(* PLC project Система умного дома.project, CODESYS CODESYS V3.5 SP17 Patch 3 *)
(* stored: creationDateTime 2026-04-06T20:38:17.5908527, modificationDateTime 2026-03-25T09:46:39.3897592 *)

TYPE E_ALERT_PRIORITY : (ALERT_PRIORITY_NONE := 0, ALERT_PRIORITY_LOW := 1, ALERT_PRIORITY_MEDIUM := 2, ALERT_PRIORITY_HIGH := 3, ALERT_PRIORITY_CRITICAL := 4) USINT;
END_TYPE

TYPE E_Debug_Log_Level : (LOG_LEVEL_MINIMAL := 0, LOG_LEVEL_NORMAL := 1, LOG_LEVEL_VERBOSE := 2, LOG_LEVEL_DEBUG := 3) USINT;
END_TYPE

TYPE E_Gateway_Command_Type : (CMD_NONE := 0, CMD_SET_SCENARIO := 1, CMD_SET_LIGHT := 2, CMD_SET_SOCKET := 3, CMD_SET_SECURITY := 4, CMD_SET_TEMP := 5, CMD_SET_VENT := 6, CMD_SET_BLINDS := 7, CMD_TELEGRAM_MSG := 8) USINT;
END_TYPE

TYPE E_Lifetime_Device_Type : (LIFETIME_DEVICE_PUMP := 1, LIFETIME_DEVICE_FAN := 2) USINT;
END_TYPE

TYPE E_Outdoor_Mode : (OUTDOOR_MODE_AUTO := 0, OUTDOOR_MODE_PARTY := 1, OUTDOOR_MODE_SECURITY := 2, OUTDOOR_MODE_ECONOMY := 3, OUTDOOR_MODE_MANUAL := 4) USINT;
END_TYPE

TYPE E_PLC_ROLE : (ROLE_UNDEFINED := 0, ROLE_ACTIVE := 1, ROLE_STANDBY := 2, ROLE_OFFLINE := 3) USINT;
END_TYPE

TYPE E_Rule_Action_Type : (ACTION_NONE := 0, ACTION_SET_FLOOR_HEATING := 1, ACTION_SET_LIGHTING_BASE := 2, ACTION_SET_LIGHTING_ACCENT := 3, ACTION_SET_SOCKET := 4, ACTION_SET_VENTILATION := 5, ACTION_SET_BLINDS := 6, ACTION_ACTIVATE_SCENARIO := 7, ACTION_TOGGLE_LIGHTING := 8, ACTION_TOGGLE_SOCKET := 9) USINT;
END_TYPE

TYPE E_Rule_Comparison : (COMP_NONE := 0, COMP_EQ := 1, COMP_GT := 2, COMP_LT := 3, COMP_GE := 4, COMP_LE := 5, COMP_IN_RANGE := 6, COMP_TRUE := 7, COMP_FALSE := 8) USINT;
END_TYPE

TYPE E_Rule_Condition_Type : (COND_NONE := 0, COND_AIR_TEMP := 1, COND_FLOOR_TEMP := 2, COND_HUMIDITY := 3, COND_CO2 := 4, COND_METHANE := 5, COND_CO := 6, COND_DOOR_WINDOW := 7, COND_FLOOD := 8, COND_SMOKE := 9, COND_MOTION := 10, COND_TIME_OF_DAY := 11, COND_DAY_OF_WEEK := 12) USINT;
END_TYPE

TYPE E_SCENARIO_TYPE : (SCENARIO_NONE := 0, SCENARIO_MORNING := 1, SCENARIO_EVENING := 2, SCENARIO_AWAY := 3, SCENARIO_PARTY := 4, SCENARIO_SLEEP := 5, SCENARIO_EMERGENCY := 6, SCENARIO_PRESENCE := 7) USINT;
END_TYPE

TYPE E_SENSOR_TYPE : (SENSOR_TYPE_NONE := 0, SENSOR_TYPE_DOOR_WINDOW := 5, SENSOR_TYPE_GLASS_BREAK := 6, SENSOR_TYPE_FLOOD := 7, SENSOR_TYPE_SMOKE := 8, SENSOR_TYPE_GAS_METHANE := 1, SENSOR_TYPE_GAS_CO := 2, SENSOR_TYPE_TEMP_FLOOR := 3, SENSOR_TYPE_TEMP_AIR := 4, SENSOR_TYPE_CO2 := 9) USINT;
END_TYPE

TYPE E_System_Operating_Mode : (MODE_NORMAL := 0, MODE_DEGRADED := 1, MODE_SAFE_STOP := 2, MODE_FREEZE_PROTECTION := 3) INT;
END_TYPE

TYPE E_System_Root_Cause : (ROOT_NONE := 0, ROOT_FIRE := 1, ROOT_GAS_LEAK := 2, ROOT_CO_WARNING := 3, ROOT_CO_CRITICAL := 4, ROOT_WATER_LEAK := 5, ROOT_IO_OFFLINE := 6, ROOT_COMM_FAULT := 7, ROOT_SENSOR_FAULT := 8, ROOT_SUBSYSTEM_FAULT := 9, ROOT_WATCHDOG_FAULT := 10) INT;
END_TYPE

TYPE E_System_Severity : (SEV_NORMAL := 0, SEV_WARNING := 1, SEV_DEGRADED := 2, SEV_CRITICAL := 3) INT;
END_TYPE

TYPE E_Trend_Parameter_Type : (TREND_PARAM_NONE := 0, TREND_PARAM_TEMP_AIR := 1, TREND_PARAM_TEMP_FLOOR := 2, TREND_PARAM_PRESSURE := 3, TREND_PARAM_PUMP_CURRENT := 4, TREND_PARAM_GAS_METHANE := 5, TREND_PARAM_GAS_CO := 6) USINT;
END_TYPE

TYPE E_TwoFactor_Method : (TF_METHOD_NONE := 0, TF_METHOD_RFID := 1, TF_METHOD_TOTP := 2, TF_METHOD_BOTH := 3) USINT;
END_TYPE

TYPE E_VALVE_TYPE : (VALVE_NC := 1, VALVE_NO := 2) USINT;
END_TYPE

TYPE E_VENTILATION_LOCATION : (VENT_LOCATION_NONE := 0, VENT_LOCATION_BASEMENT_GAME_ROOM := 1, VENT_LOCATION_BASEMENT_GYM := 2, VENT_LOCATION_BASEMENT_BOILER_ROOM := 3, VENT_LOCATION_BATHROOM_1F := 4, VENT_LOCATION_BATHROOM_2F := 5, VENT_LOCATION_MASTER_BATHROOM := 6, VENT_LOCATION_LAUNDRY := 7, VENT_LOCATION_KITCHEN := 8) USINT;
END_TYPE

TYPE E_VENTILATION_UNIT_TYPE : (VENTILATION_TYPE_NONE := 0, VENTILATION_TYPE_SUPPLY := 1, VENTILATION_TYPE_EXHAUST := 2) USINT;
END_TYPE

TYPE E_Valve_Test_Result : (TEST_RESULT_NONE := 0, TEST_RESULT_PASSED := 1, TEST_RESULT_CURRENT_DEVIATION := 2, TEST_RESULT_TIME_DEVIATION := 3, TEST_RESULT_STALL := 4, TEST_RESULT_LIMIT_SWITCH_FAIL := 5, TEST_RESULT_ABORTED := 6) USINT;
END_TYPE

TYPE E_WEATHER_COMPENSATION_METHOD : (WEATHER_COMP_NONE := 0, WEATHER_COMP_OUTDOOR_RESET := 1) USINT;
END_TYPE

TYPE E_Zone_Access_Level : (ZONE_ACCESS_NONE := 0, ZONE_ACCESS_VIEW := 1, ZONE_ACCESS_CONTROL := 2, ZONE_ACCESS_CONFIG := 3, ZONE_ACCESS_FULL := 4) USINT;
END_TYPE

TYPE ST_Alarm_Record : STRUCT
  ID : UDINT;
  Timestamp_MS : UDINT;
  Source : STRING(20);
  Source_ID : BYTE;
  Message : STRING(100);
  Severity : E_ALERT_PRIORITY;
  Is_Active : BOOL;
  Is_Acknowledged : BOOL;
END_STRUCT;
END_TYPE

TYPE ST_Astro_Time : STRUCT
  sunrise_ms : UDINT := 0;
  sunset_ms : UDINT := 0;
  is_daylight : BOOL := FALSE;
END_STRUCT;
END_TYPE

TYPE ST_BlackBox_Record : STRUCT
  Timestamp : UDINT;
  Gas_Methane_LEL : REAL;
  Gas_CO_PPM : REAL;
  Flood_Active : BOOL;
  Fire_Active : BOOL;
  Valve_Gas_Status : BYTE;
  Valve_Water_Status : BYTE;
  PLC_Active_ID : BYTE;
  System_Mode : BYTE;
  First_Fault_Type : BYTE;
  First_Fault_Source : BYTE;
  First_Fault_Active : BOOL;
  System_Severity : BYTE;
  Root_Cause : BYTE;
  Watchdog_Fault : BOOL;
END_STRUCT;
END_TYPE

TYPE ST_BlackBox_Snapshot_V2 : STRUCT
  Gas_Alarm : BOOL;
  Fire_Alarm : BOOL;
  Flood_Alarm : BOOL;
  First_Fault_Type : BYTE;
  First_Fault_Source : BYTE;
END_STRUCT;
END_TYPE

TYPE ST_Blinds_Command_V2 : STRUCT
  Position_Setpoint : BYTE;
END_STRUCT;
END_TYPE

TYPE ST_Blinds_State_V2 : STRUCT
  Position_Actual : BYTE;
END_STRUCT;
END_TYPE

TYPE ST_Boiler_Status : STRUCT
  Active : BOOL;
  Running : BOOL;
  Warning : BOOL;
  Error : BOOL;
  Error_ID : WORD;
  Power_Percent : REAL;
  Current_Power : REAL;
  Work_Seconds : UDINT;
  Work_Hours : REAL;
  Resource_Percent : REAL := 100.0;
  Last_Start : DT;
END_STRUCT;
END_TYPE

TYPE ST_Component_Maintenance : STRUCT
  Is_Faulty : BOOL;
  Is_In_Maintenance : BOOL;
  Fallback_Value : REAL;
  Use_Last_Good_Value : BOOL;
END_STRUCT;
END_TYPE

TYPE ST_DHW_Command_V2 : STRUCT
  Pump_Enable : REAL;
END_STRUCT;
END_TYPE

TYPE ST_DHW_Config : STRUCT
  Target_Temp : REAL := 55.0;
  Hysteresis : REAL := 2.0;
  Circulation_Schedule_Enabled : BOOL := TRUE;
  Circulation_Start : TOD := TOD#06:00;
  Circulation_End : TOD := TOD#23:00;
  Night_Mode_Enabled : BOOL := TRUE;
  Anti_Legionella_Enabled : BOOL := TRUE;
  Anti_Legionella_Day : UINT := 7;
  Degraded_Target_Delta : REAL := 5.0;
END_STRUCT;
END_TYPE

TYPE ST_DHW_State_V2 : STRUCT
  Tank_Temp : REAL;
  Supply_Temp : REAL;
END_STRUCT;
END_TYPE

TYPE ST_DHW_Status : STRUCT
  Temp : REAL;
  Pressure : REAL;
  Heating_Pump_On : BOOL;
  Circ_Pump_On : BOOL;
  Warning : BOOL;
  Error : BOOL;
  Error_ID : WORD;
END_STRUCT;
END_TYPE

TYPE ST_Debug_Log_Record : STRUCT
  timestamp_ms : UDINT;
  level : BYTE;
  source_id : BYTE;
  event_code : WORD;
  value_int : UDINT;
  value_real : REAL;
  text : STRING(80);
  crc32 : DWORD;
END_STRUCT;
END_TYPE

TYPE ST_Debug_Logger_Config : STRUCT
  enabled : BOOL;
  sampling_period_ms : UDINT := GVL_CONSTANTS.C_MS_IN_SECOND;
END_STRUCT;
END_TYPE

TYPE ST_Device_Health : STRUCT
  Health_Score : BYTE := 100;
  Total_Runtime_Hours : UDINT;
  Starts_Count : UDINT;
  Last_Start_Current : REAL;
  Avg_Start_Current : REAL;
  Sample_Count : UDINT;
  Current_Sum : REAL;
  Maintenance_Required : BOOL;
  Warning_Message : STRING(50);
END_STRUCT;
END_TYPE

TYPE ST_Flood_Config : STRUCT
  Emergency_Two_Stage_Enabled : BOOL := TRUE;
  Valve_Test_Period_Days : UINT := 7;
  Current_Threshold_MA : REAL := 500.0;
  sensor_to_valve_map : ARRAY[1..GVL_CONSTANTS.C_MAX_FLOOD_SENSORS] OF INT := [1, 1, 1, 1, 2, 2, 2, 2, 3, 3, 3, 3];
END_STRUCT;
END_TYPE

TYPE ST_Flood_Global_Config : STRUCT
  valve_types : ARRAY[1..GVL_CONSTANTS.C_MAX_FLOOD_VALVES] OF E_VALVE_TYPE := [GVL_CONSTANTS.C_MAX_FLOOD_VALVES(E_VALVE_TYPE.VALVE_NC)];
  sensor_to_valve_map : ARRAY[1..GVL_CONSTANTS.C_MAX_FLOOD_SENSORS] OF BYTE := [1, 1, 1, 2, 2, 2, 2, 0, 0, 0];
  min_duration_ms : UDINT := 5000;
  warning_duration_ms : UDINT := 30000;
END_STRUCT;
END_TYPE

TYPE ST_FloorHeating_Circuit_Config : STRUCT
  circuit_id : BYTE := 0;
  zone : BYTE := 0;
  manifold_id : BYTE := 1;
  sensor_id : BYTE := 1;
  valve_id : BYTE := 1;
  control_type : BYTE := 1;
  design_temp : REAL := 35.0;
  min_temp : REAL := 20.0;
  max_temp : REAL := 45.0;
  pid_kp : REAL := 2.0;
  pwm_period_s : UINT := 600;
END_STRUCT;
END_TYPE

TYPE ST_FloorHeating_Global_Config : STRUCT
  enable_floor_heating : BOOL := TRUE;
  anti_freeze_temp : REAL := 7.0;
  overheat_temp : REAL := 45.0;
  weather_compensation_enabled : BOOL := TRUE;
  total_circuits : BYTE := 16;
END_STRUCT;
END_TYPE

TYPE ST_FloorHeating_Manifold_Config : STRUCT
  manifold_id : BYTE;
  location : STRING(30);
  nominal_flow : REAL;
  enable_pump : BOOL;
  circuits : ARRAY[1..GVL_CONSTANTS.C_MAX_CIRCUITS_PER_MANIFOLD] OF ST_FloorHeating_Circuit_Config;
END_STRUCT;
END_TYPE

TYPE ST_Gas_Valve_Configuration : STRUCT
  valve_id : BYTE := 0;
  valve_type : E_VALVE_TYPE := E_VALVE_TYPE.VALVE_NC;
  close_time_seconds : UDINT := 10;
  open_time_seconds : UDINT := 10;
  emergency_open_allowed : BOOL := FALSE;
END_STRUCT;
END_TYPE

TYPE ST_Gateway_Command : STRUCT
  command_id : UDINT;
  timestamp_ms : UDINT;
  operator_id : STRING(10);
  command_type : E_Gateway_Command_Type;
  target_zone : BYTE;
  target_value : REAL;
  target_on_off : BOOL;
  target_scenario : E_SCENARIO_TYPE;
  target_armed : BOOL;
  target_pin : STRING(4);
  target_2fa_code : STRING(6);
  telegram_msg : STRING(200);
  source_ip : STRING(15);
  crc32 : DWORD;
END_STRUCT;
END_TYPE

TYPE ST_Heating_Command_V2 : STRUCT
  Valve_Position_Setpoint : REAL;
END_STRUCT;
END_TYPE

TYPE ST_Heating_Config : STRUCT
  Weather_Comp_Enabled : BOOL := TRUE;
  Weather_Coef : REAL := 0.1;
  Freeze_Threshold : REAL := 7.0;
  Overheat_Threshold : REAL := 45.0;
  Night_Reduction : REAL := 3.0;
  Target_Floor_Temp : REAL := 28.0;
  Target_Room_Temp : REAL := 22.0;
  Hysteresis : REAL := 0.5;
END_STRUCT;
END_TYPE

TYPE ST_Heating_State_V2 : STRUCT
  Room_Temp : REAL;
  Supply_Temp : REAL;
END_STRUCT;
END_TYPE

TYPE ST_History_Event_V2 : STRUCT
  Event_Code : UINT;
  Event_Value : REAL;
END_STRUCT;
END_TYPE

TYPE ST_History_Record : STRUCT
  timestamp_ms : UDINT := 0;
  event_code : WORD := 0;
  event_value : REAL := 0.0;
  unit : BYTE := 0;
  zone_id : BYTE := 0;
  operator_id : STRING(10) := '';
  priority : E_ALERT_PRIORITY := E_ALERT_PRIORITY.ALERT_PRIORITY_NONE;
END_STRUCT;
END_TYPE

TYPE ST_Lifetime_Status : STRUCT
  device_id : BYTE;
  runtime_hours : UDINT;
  start_count : UDINT;
  remaining_hours : UDINT;
  remaining_percent : BYTE;
  maintenance_required : BOOL;
  last_calc_timestamp : UDINT;
END_STRUCT;
END_TYPE

TYPE ST_Lighting_Command_V2 : STRUCT
  Brightness_Setpoint : REAL;
END_STRUCT;
END_TYPE

TYPE ST_Lighting_State_V2 : STRUCT
  Brightness_Actual : REAL;
  Motion_Active : BOOL;
END_STRUCT;
END_TYPE

TYPE ST_Maintenance_Access_Config : STRUCT
  maintenance_enabled : BOOL := FALSE;
  max_duration_minutes : UDINT := 60;
  requires_two_person : BOOL := TRUE;
  access_level_required : BYTE := 2;
END_STRUCT;
END_TYPE

TYPE ST_Manifold_Status : STRUCT
  Pump_On : BOOL;
  Pump_Current : REAL;
  Pressure : REAL;
  Temp_Supply : REAL;
  Temp_Return : REAL;
  Valve_Pos : REAL;
  Error : BOOL;
  Error_ID : WORD;
  Health : ST_Device_Health;
END_STRUCT;
END_TYPE

TYPE ST_Operator_Zone_Rights : STRUCT
  operator_id : STRING(10);
  global_access_level : BYTE := 0;
  zone_masks : DWORD;
  last_modified : UDINT;
END_STRUCT;
END_TYPE

TYPE ST_Outdoor_Zone_Config : STRUCT
  zone_id : BYTE := 0;
  lighting_circuit_id : BYTE := 0;
  auto_enabled : BOOL := TRUE;
  party_mode_enabled : BOOL := FALSE;
END_STRUCT;
END_TYPE

TYPE ST_Owen_Analog_Value : STRUCT
  rValue : REAL;
  uiCycleTime : UINT;
  wStatus : WORD;
END_STRUCT;
END_TYPE

TYPE ST_Rule : STRUCT
  Action_Type : INT;
  Action_Target_ID : INT;
  Action_Value : REAL;
  Condition_Type : INT;
  Condition_Target_ID : INT;
  Condition_Op : INT;
  Condition_Value : REAL;
  Condition_Value_Max : REAL;
END_STRUCT;
END_TYPE

TYPE ST_Rule_Action : STRUCT
  Active : BOOL;
  Triggered : BOOL;
  Action_Type : E_Rule_Action_Type;
  Target_ID : BYTE;
  Value : REAL;
END_STRUCT;
END_TYPE

TYPE ST_Scenario_Config : STRUCT
  scenario_id : E_SCENARIO_TYPE;
  lighting_level_base : BYTE := 100;
  lighting_level_accent : BYTE := 100;
  floor_heating_adjust_celsius : REAL := 0.0;
  ventilation_speed_percent : BYTE := 50;
  sockets_enabled : BOOL := TRUE;
  blinds_position_percent : BYTE := 0;
  Presence_Simulation_Enabled : BOOL := FALSE;
END_STRUCT;
END_TYPE

TYPE ST_Scenario_Transition_Config : STRUCT
  current_scenario : E_SCENARIO_TYPE;
  target_scenario : E_SCENARIO_TYPE;
  min_duration_minutes : UDINT := 5;
  transition_allowed : BOOL := FALSE;
END_STRUCT;
END_TYPE

TYPE ST_Security_Global_Config : STRUCT
  PIN_Code : STRING(4) := '1234';
  Phones : ARRAY[1..GVL_CONSTANTS.C_MAX_SECURITY_PHONES] OF STRING(15);
  entry_delay_seconds : UDINT := 30;
  exit_delay_seconds : UDINT := 60;
  alarm_duration_seconds : UDINT := 180;
  two_person_timeout_seconds : UDINT := 120;
  max_access_attempts : BYTE := 3;
  auto_arm_enabled : BOOL := FALSE;
  auto_arm_time_ms : UDINT := 0;
  enable_2fa : BOOL := TRUE;
  gate_open_pulse_ms : UDINT := GVL_CONSTANTS.C_MS_IN_SECOND;
  wicket_open_pulse_ms : UDINT := GVL_CONSTANTS.C_MS_IN_SECOND;
  lock_open_pulse_ms : UDINT := GVL_CONSTANTS.C_MS_IN_SECOND;
  lock_close_pulse_ms : UDINT := GVL_CONSTANTS.C_MS_IN_SECOND;
  bypass_motion : ARRAY[1..16] OF BOOL;
  bypass_doors : ARRAY[1..GVL_CONSTANTS.C_MAX_DOOR_SENSORS] OF BOOL;
  bypass_windows : ARRAY[1..16] OF BOOL;
END_STRUCT;
END_TYPE

TYPE ST_Security_Zone_State : STRUCT
  Armed : BOOL;
  Alarm : BOOL;
  Bypassed : BOOL;
  Last_Trigger_Time : DT;
  Trigger_Count : UINT;
END_STRUCT;
END_TYPE

TYPE ST_Sensor_Calibration_Record : STRUCT
  sensor_id : UDINT := 0;
  sensor_type : E_SENSOR_TYPE;
  zone_id : BYTE := 0;
  offset : REAL := 0.0;
  multiplier : REAL := 1.0;
  last_calibration_timestamp : UDINT := 0;
  verification_passed : BOOL := FALSE;
END_STRUCT;
END_TYPE

TYPE ST_Socket_Command_V2 : STRUCT
  Target_State : BOOL;
END_STRUCT;
END_TYPE

TYPE ST_Socket_State_V2 : STRUCT
  Is_On : BOOL;
  Safety_Blocked : BOOL;
END_STRUCT;
END_TYPE

TYPE ST_State_Snapshot : STRUCT
  timestamp_ms : UDINT := 0;
  operator_id : STRING(10) := '';
  scenario_id : E_SCENARIO_TYPE := E_SCENARIO_TYPE.SCENARIO_NONE;
  lighting_levels : ARRAY[1..GVL_CONSTANTS.C_MAX_LIGHTING_ZONES] OF BYTE;
  floor_heating_setpoints : ARRAY[1..GVL_CONSTANTS.C_MAX_HEATING_CIRCUITS] OF REAL;
  alarm_active : BOOL := FALSE;
  crc32 : DWORD := 0;
END_STRUCT;
END_TYPE

TYPE ST_System_Diagnostics : STRUCT
  Freeze_Hardware_Event_Pending : BOOL;
  Freeze_Hardware_Event_Text : STRING(200);
  Backup_Pump_Fault : BOOL;
  Electric_Heater_Fault : BOOL;
  Backup_Pump_Recovered_After_Retry : BOOL;
  Electric_Heater_Recovered_After_Retry : BOOL;
  Backup_Pump_Out_Of_Service : BOOL;
  Electric_Heater_Out_Of_Service : BOOL;
  Pump_Exercise_Active : BOOL;
  Pump_Exercise_Failed : BOOL;
  Pump_Exercise_Last_Equipment : STRING(80);
  Pump_Exercise_Last_Result : STRING(120);
  Pump_Exercise_No_Feedback_Count : INT;
  Manifold_Pump_Exercise_Count : ARRAY[1..GVL_CONSTANTS.C_MAX_MANIFOLDS] OF UDINT;
  DHW_Heating_Pump_Exercise_Count : UDINT;
  DHW_Circ_Pump_Exercise_Count : UDINT;
  Backup_Pump_Exercise_Count : UDINT;
  Pump_Exercise_Event_Seq : UDINT;
  Pump_Exercise_Journal_1 : STRING(200);
  Pump_Exercise_Journal_2 : STRING(200);
  Pump_Exercise_Journal_3 : STRING(200);
  Pump_Exercise_Journal_Last_Seq : UDINT;
  Pump_Maintenance_Required : BOOL;
  Pump_Maintenance_Warning : BOOL;
  Manifold_Pump_Out_Of_Service : ARRAY[1..GVL_CONSTANTS.C_MAX_MANIFOLDS] OF BOOL;
  DHW_Heating_Pump_Out_Of_Service : BOOL;
  DHW_Circ_Pump_Out_Of_Service : BOOL;
  Maintenance_Last_Action : STRING(120);
  Operator_Action_Blocked : BOOL;
  Operator_Block_Reason : STRING(160);
  Operator_Last_Forbidden_Action : STRING(160);
  Operator_Journal_1 : STRING(200);
  Operator_Journal_2 : STRING(200);
  Operator_Journal_3 : STRING(200);
  Operator_Journal_Event_Seq : UDINT;
  Operator_Journal_Last_Seq : UDINT;
  Dangerous_Action_Pending_Confirm : BOOL;
  Dangerous_Action_Confirm_Text : STRING(160);
  Dangerous_Action_Confirm_Deadline_MS : UDINT;
  User_Access_Level_Active : INT;
  User_Access_Denied : BOOL;
  User_Access_Deny_Reason : STRING(160);
  Valve_Test_Mode_Active : BOOL;
  Valve_Test_Deadline_MS : UDINT;
  Valve_Test_Remaining_MS : UDINT;
  Valve_Test_Validation_OK : BOOL;
  Valve_Test_Validation_Text : STRING(160);
  Valve_Test_Forced_Close : BOOL;
  Water_Valve_Test_Mode_Active : BOOL;
  Water_Valve_Test_Deadline_MS : UDINT;
  Water_Valve_Test_Remaining_MS : UDINT;
  Water_Valve_Test_Validation_OK : BOOL;
  Water_Valve_Test_Validation_Text : STRING(160);
  Water_Valve_Test_Forced_Close : BOOL;
  Gas_Valve_Test_Mode_Active : BOOL;
  Gas_Valve_Test_Deadline_MS : UDINT;
  Gas_Valve_Test_Remaining_MS : UDINT;
  Gas_Valve_Test_Validation_OK : BOOL;
  Gas_Valve_Test_Validation_Text : STRING(160);
  Gas_Valve_Test_Forced_Close : BOOL;
  Active_Leak_Sensor_Index : INT;
  Active_Gas_Sensor_Index : INT;
  Active_Leak_Zone_Name : STRING(80);
  Active_Gas_Zone_Name : STRING(80);
  Water_Valve_Test_Context : STRING(160);
  Gas_Valve_Test_Context : STRING(160);
  Water_Recovery_Target_Zone_Index : INT;
  Gas_Recovery_Target_Zone_Index : INT;
  Water_Recovery_Selective_Allowed : BOOL;
  Gas_Recovery_Selective_Allowed : BOOL;
  Water_Recovery_Selective_Text : STRING(160);
  Gas_Recovery_Selective_Text : STRING(160);
  Water_Recovery_Physical_Active : BOOL;
  Water_Recovery_Physical_Zone_Name : STRING(80);
  Water_Zone_Open_Fault : ARRAY[1..32] OF BOOL;
  Water_Zone_Close_Fault : ARRAY[1..32] OF BOOL;
  Water_Valve_Exercise_Last_Zone : INT;
  Water_Valve_Exercise_Last_Result : STRING(160);
  Water_Zone_Critical_Close_Fault : ARRAY[1..32] OF BOOL;
  Water_Close_Fault_Active : BOOL;
  Water_Close_Fault_Zone_Name : STRING(80);
  Water_Close_Fault_Text : STRING(200);
  Water_Zone_Close_Retry_Active : ARRAY[1..32] OF BOOL;
  Water_Zone_Close_Retry_Count : ARRAY[1..32] OF INT;
  Water_Zone_Close_Recovered_After_Retry : ARRAY[1..32] OF BOOL;
  Water_Localization_Failed : BOOL;
  Water_Main_Shutdown_Recommended : BOOL;
  Water_Escalation_Text : STRING(200);
  Alarm_Event_Pulse : BOOL;
  Alarm_Event_Code : UDINT;
  Alarm_Event_Value : REAL;
  Sensor_Fault : BOOL;
  IO_Offline : BOOL;
  Subsystem_Degraded : BOOL;
END_STRUCT;
END_TYPE

TYPE ST_System_State_Snapshot : STRUCT
  System_Time_MS : UDINT;
  Current_Scenario : E_SCENARIO_TYPE;
  Security_Armed : BOOL;
  Active_Alarms : INT;
  Zone_Valves : ARRAY[1..8] OF BOOL;
  Manifold_Pumps : ARRAY[1..GVL_CONSTANTS.C_MAX_MANIFOLDS] OF BOOL;
  Lighting_States : ARRAY[1..32] OF BYTE;
  Blinds_Positions : ARRAY[1..GVL_CONSTANTS.C_MAX_BLINDS] OF BYTE;
  Socket_States : ARRAY[1..GVL_CONSTANTS.C_MAX_SOCKETS] OF BOOL;
  Gas_Valve_Closed : BOOL;
  Water_Valves_Closed : BOOL;
  Version : UDINT;
END_STRUCT;
END_TYPE

TYPE ST_System_State_Summary : STRUCT
  Outdoor_Temp : REAL;
  Indoor_Temp : ARRAY[1..GVL_CONSTANTS.C_MAX_CLIMATE_ZONES] OF REAL;
  Floor_Temps : ARRAY[1..GVL_CONSTANTS.C_MAX_HEATING_CIRCUITS] OF REAL;
  Humidity : ARRAY[1..GVL_CONSTANTS.C_MAX_HUMIDITY_SENSORS] OF REAL;
  CO2 : ARRAY[1..GVL_CONSTANTS.C_MAX_CO2_SENSORS] OF REAL;
  Gas_Alarm : BOOL;
  Flood_Alarm : BOOL;
  Fire_Alarm : BOOL;
  Security_Alarm : BOOL;
  Security_Armed : BOOL;
END_STRUCT;
END_TYPE

TYPE ST_Tariff_Config : STRUCT
  Enabled : BOOL := FALSE;
  Night_Start_Hour : UINT := 23;
  Night_End_Hour : UINT := 7;
  Boost_Delta : REAL := 2.0;
END_STRUCT;
END_TYPE

TYPE ST_Trend_Config : STRUCT
  param_type : BYTE;
  zone_id : BYTE;
  enabled : BOOL;
  deviation_threshold_percent : REAL := 10.0;
  history_days : UDINT := 7;
END_STRUCT;
END_TYPE

TYPE ST_Trend_Data : STRUCT
  config : ST_Trend_Config;
  record_count : UDINT;
  write_index : UDINT;
  sum_values : REAL;
  values : ARRAY[1..100] OF REAL;
  timestamps : ARRAY[1..100] OF UDINT;
  crc32 : DWORD;
END_STRUCT;
END_TYPE

TYPE ST_Trend_Header : STRUCT
  parameter_type : BYTE;
  zone_id : BYTE := 0;
  records_count : UDINT := 0;
  average_value : REAL := 0.0;
  min_value : REAL := 0.0;
  max_value : REAL := 0.0;
END_STRUCT;
END_TYPE

TYPE ST_Trend_History_Record : STRUCT
  timestamp_ms : UDINT := 0;
  value : REAL := 0.0;
END_STRUCT;
END_TYPE

TYPE ST_TwoFactor_Auth_State : STRUCT
  Auth_Method : E_TwoFactor_Method;
  is_pending : BOOL;
  Attempts_Left : UINT;
  Time_Left_S : UINT;
  Is_Success : BOOL;
  Is_Locked : BOOL;
END_STRUCT;
END_TYPE

TYPE ST_TwoFactor_Data : STRUCT
  operator_id : STRING(10);
  AuthMethod : BYTE;
  rfid_tag : STRING(20);
  totp_secret : STRING(32);
  last_modified : UDINT;
END_STRUCT;
END_TYPE

TYPE ST_User_Rule : STRUCT
  Enabled : BOOL;
  Condition_Type : E_Rule_Condition_Type;
  Condition_Target_ID : BYTE;
  Condition_Op : E_Rule_Comparison;
  Condition_Value : REAL;
  Condition_Value_Max : REAL;
  Action_Target_ID : BYTE;
  Action_Value : REAL;
  Action_Type : E_Rule_Action_Type;
  Priority : BYTE;
END_STRUCT;
END_TYPE

TYPE ST_Valve_Test_Config : STRUCT
  valve_id : BYTE := 0;
  test_interval_days : UDINT := 7;
  Nominal_Current : REAL := 0.5;
  nominal_close_time_sec : REAL := 10.0;
  enabled : BOOL := TRUE;
END_STRUCT;
END_TYPE

TYPE ST_Ventilation_Command_V2 : STRUCT
  Fan_Speed_Setpoint : REAL;
END_STRUCT;
END_TYPE

TYPE ST_Ventilation_Config : STRUCT
  CO2_Threshold : REAL := 800.0;
  Humidity_Threshold : REAL := 65.0;
  Night_Mode_Start : TOD := TOD#23:00;
  Night_Mode_End : TOD := TOD#07:00;
END_STRUCT;
END_TYPE

TYPE ST_Ventilation_Global_Config : STRUCT
  enable_ventilation : BOOL := TRUE;
  total_units : BYTE := 8;
  default_supply_speed : BYTE := 40;
  default_exhaust_speed : BYTE := 40;
  Degraded_Exhaust_Limit : BYTE := 30;
  Scenario_Modes : ARRAY[1..GVL_CONSTANTS.C_MAX_SCENARIOS] OF ST_Ventilation_Scenario_Mode;
  wet_zone_to_exhaust_map : ARRAY[1..GVL_CONSTANTS.C_MAX_WET_ZONES] OF INT := [2, 3, 4, 5];
  pv3_exhaust_index : INT := 3;
END_STRUCT;
END_TYPE

TYPE ST_Ventilation_Scenario_Mode : STRUCT
  Scenario_ID : BYTE;
  Scenario_Priority : BYTE;
  Fire_Alarm : BOOL;
  Methane_Alarm : BOOL;
  Smoke_Detected : BOOL;
  Exhaust_Modes : ARRAY[1..GVL_CONSTANTS.C_MAX_EXHAUST_FANS] OF BYTE;
  Supply_Modes : ARRAY[1..GVL_CONSTANTS.C_MAX_SUPPLY_FANS] OF BYTE;
  Base_Fan_Speed : BYTE := 50;
  Target_Temp : REAL := 22.0;
END_STRUCT;
END_TYPE

TYPE ST_Ventilation_State_V2 : STRUCT
  Supply_Temp : REAL;
END_STRUCT;
END_TYPE

TYPE ST_Ventilation_Unit : STRUCT
  Enabled : BOOL;
  Speed_Percent : REAL;
  Filter_Dirty : BOOL;
  Error : BOOL;
  Mode : BYTE;
END_STRUCT;
END_TYPE

TYPE ST_Ventilation_Unit_Config : STRUCT
  unit_id : BYTE := 0;
  unit_type : E_VENTILATION_UNIT_TYPE;
  location : E_VENTILATION_LOCATION;
  min_speed : BYTE := 20;
  max_speed : BYTE := 100;
  Threshold_Hum : REAL := 65.0;
  has_smoke_detector : BOOL := FALSE;
END_STRUCT;
END_TYPE

TYPE ST_Zone_Sensors : STRUCT
  Temp_Room : REAL;
  Temp_Floor : REAL;
  Motion_Active : BOOL;
  Switch_Physical : BOOL;
  Light_State : BOOL;
  Maintenance : ST_Component_Maintenance;
END_STRUCT;
END_TYPE

{attribute 'qualified_only'}
VAR_GLOBAL  (* GVL_CONFIG *)
  G_Heating_Config : ST_Heating_Config;  (* Настройки системы отопления *)
  G_Ventilation_Config : ST_Ventilation_Config;  (* Настройки системы вентиляции *)
  G_DHW_Config : ST_DHW_Config;  (* Настройки горячего водоснабжения *)
  G_Security_Config : ST_Security_Global_Config;  (* Настройки системы безопасности *)
  G_Flood_Config : ST_Flood_Config;  (* Настройки системы защиты от протечек *)
  G_HMI_FloorHeating_Configs : ARRAY[1..8] OF ST_FloorHeating_Circuit_Config;  (* Конфигурации контуров теплого пола *)
  G_Wet_Zone_Map : ARRAY[1..32] OF BOOL;  (* Карта мокрых зон (TRUE = мокрая зона) *)
  G_HMI_Tariff_Settings : ST_Tariff_Config;  (* Настройки тарифов *)
  G_HMI_Vent_Global_Config : ST_Ventilation_Global_Config;  (* Глобальные настройки вентиляции *)
  G_HMI_Vent_Unit_Configs : ARRAY[1..GVL_CONSTANTS.C_MAX_VENT_UNITS] OF ST_Ventilation_Unit_Config;  (* Конфигурации отдельных вентустановок *)
  G_HMI_Scenario_Configs : ARRAY[1..GVL_CONSTANTS.C_MAX_SCENARIOS] OF ST_Scenario_Config;  (* Конфигурации сценариев *)
  G_HMI_Outdoor_Configs : ARRAY[1..GVL_CONSTANTS.C_MAX_OUTDOOR_ZONES] OF ST_Outdoor_Zone_Config;  (* Конфигурации зон уличного освещения *)
  G_HMI_Flood_Config : ST_Flood_Global_Config;  (* Глобальные настройки защиты от протечек *)
  G_HMI_Gas_Config : ST_Gas_Valve_Configuration;  (* Конфигурация системы газового контроля *)
  G_HMI_Sensor_Calibrations : ARRAY[1..GVL_CONSTANTS.C_MAX_CALIBRATIONS] OF ST_Sensor_Calibration_Record;  (* Данные калибровки датчиков *)
  G_HMI_User_Rules : ARRAY[1..GVL_CONSTANTS.C_MAX_RULES] OF ST_User_Rule;  (* Пользовательские правила (Rule Engine) *)
  G_Valve_Test_Config : ARRAY[1..GVL_CONSTANTS.C_MAX_MANIFOLDS] OF ST_Valve_Test_Config;
  G_HMI_Cleaning_Mode_Active : ARRAY[1..GVL_CONSTANTS.C_MAX_CLEANING_MODES] OF BOOL;  (* Режим уборки активен *)
  G_HMI_Cleaning_Mode_TimeLeft : ARRAY[1..GVL_CONSTANTS.C_MAX_CLEANING_MODES] OF UINT;  (* Оставшееся время режима уборки *)
  G_HMI_Admin_2FA_Enabled : BOOL := FALSE;  (* Включена ли 2FA для ADMIN *)
  G_HMI_Current_Operator_Factor2_Done : BOOL;  (* Второй фактор пройден *)
  G_HMI_Current_Operator_ID : STRING(10);  (* ID текущего оператора *)
  G_HMI_Manual_Gas_Valve_Open : BOOL;  (* Ручное открытие газового клапана *)
  G_HMI_Manual_Gas_Valve_Time : UDINT := 5;  (* Время ручного открытия *)
  G_HMI_Manual_Gas_Valve_TimeLeft : UDINT;  (* Оставшееся время ручного открытия *)
  G_HMI_Apply_Settings : BOOL;  (* Команда: Применить настройки *)
  G_HMI_Mute_Alarm : BOOL;  (* Команда: Временное отключение сирены *)
  G_HMI_Ack_Alarms : BOOL;  (* Команда: Квитировать все тревоги *)
  G_HMI_Gate_Open_Req : BOOL;  (* Запрос на открытие въездных ворот *)
  G_HMI_Wicket_Open_Req : BOOL;  (* Запрос на открытие калитки *)
  G_HMI_Lock_1_Open_Req : BOOL;  (* Разблокировка основного замка *)
  G_HMI_Lock_1_Close_Req : BOOL;  (* Блокировка основного замка *)
  G_HMI_Lock_2_Open_Req : BOOL;  (* Разблокировка доп. замка *)
  G_HMI_Lock_2_Close_Req : BOOL;  (* Блокировка доп. замка *)
  G_HMI_Language : BYTE := 0;  (* 0=RU, 1=EN *)
  G_HMI_Brightness : BYTE := 80;
  G_HMI_Screen_Saver_Timeout : UDINT := 300;  (* сек *)
  G_Allowed_IPs : ARRAY[1..GVL_CONSTANTS.C_MAX_ALLOWED_IPS] OF STRING(15) := ['192.168.1.100', '192.168.1.101', '127.0.0.1', '', ''];  (* Разрешенные IP-адреса для шлюза *)
  G_Backup_Circulation_Pump_In_Service : BOOL := TRUE;  (* Резервный насос доступен для логики *)
  G_Electric_Heater_In_Service : BOOL := TRUE;  (* Электронагреватель доступен для логики *)
  G_Freeze_Hardware_Retry_Count : INT := 2;  (* Количество повторных попыток для anti-freeze hardware *)
  G_Freeze_Hardware_Retry_Delay_MS : UDINT := 5000;  (* Задержка между попытками повторного пуска *)
  G_Pump_Exercise_Enabled : BOOL := TRUE;  (* Разрешение периодической прокрутки насосов после простоя *)
  G_Pump_Exercise_Interval_MS : UDINT := 604800000;  (* 7 суток *)
  G_Pump_Exercise_Duration_MS : UDINT := 30000;  (* 30 сек *)
  G_Manifold_Pump_In_Service : ARRAY[1..GVL_CONSTANTS.C_MAX_MANIFOLDS] OF BOOL := [TRUE, TRUE, TRUE, TRUE, TRUE];
  G_DHW_Heating_Pump_In_Service : BOOL := TRUE;
  G_DHW_Circ_Pump_In_Service : BOOL := TRUE;
  G_Water_Valve_Exercise_Enabled : BOOL := TRUE;
  G_Water_Valve_Exercise_Interval_MS : UDINT := 604800000;
  G_Water_Valve_Exercise_Duration_MS : UDINT := 15000;
  G_Water_Valve_Exercise_Window_Start : TOD := TOD#04:00;
  G_Water_Valve_Exercise_Window_End : TOD := TOD#05:00;
  G_Water_Valve_Close_Retry_Count : INT := 2;
  G_Water_Valve_Close_Retry_Delay_MS : UDINT := 3000;
  G_FloorTemp_Map : ARRAY[1..8] OF INT := [1, 2, 3, 4, 5, 6, 7, 8];
  G_RoomTemp_Map : ARRAY[1..16] OF INT := [1, 2, 3, 4, 5, 6, 7, 8, 9, 10, 11, 12, 13, 14, 15, 16];
  G_Door_Map : ARRAY[1..GVL_CONSTANTS.C_MAX_DOOR_SENSORS] OF INT := [1, 2, 3, 4, 5, 6, 7, 8];
  G_Window_Map : ARRAY[1..16] OF INT := [9, 10, 11, 12, 13, 14, 15, 16, 17, 18, 19, 20, 21, 22, 23, 24];
  C_MAX_LIGHT_ZONES : INT := 32;  (* fallback if not defined elsewhere *)
  G_Evac_Exit_Zones : ARRAY[1..32] OF BOOL;  (* зоны-выходы (TRUE = выход) *)
  G_Evac_Smoke_Zone_Map : ARRAY[1..GVL_CONSTANTS.C_MAX_SMOKE_SENSORS] OF INT;  (* Привязка дымовых датчиков к зонам эвакуации *)
  G_Evac_Leak_Zone_Map : ARRAY[1..GVL_CONSTANTS.C_MAX_FLOOD_SENSORS] OF INT;  (* Привязка датчиков протечки к зонам эвакуации *)
  G_Evac_Gas_Zone_Map : ARRAY[1..GVL_CONSTANTS.C_MAX_METHANE_SENSORS] OF INT;  (* Привязка газовых датчиков к зонам эвакуации *)
  G_Evac_Zone_Names : ARRAY[1..32] OF STRING(80);  (* Человекочитаемые имена зон (помещения/крыло/этаж/сторона) *)
END_VAR

{attribute 'qualified_only'}
VAR_GLOBAL  (* GVL_GATEWAY *)
  G_Gateway_Command : ST_Gateway_Command;
  G_Gateway_Command_Received : BOOL;
  G_Gateway_Send_2FA : BOOL;
  G_Gateway_2FA_Code : STRING(6);
  G_Gateway_Telegram_Msg : STRING(200);
  G_Gateway_Send_Telegram : BOOL;
  G_Gateway_HMI_Status_Message : STRING(200);
  G_Gateway_Ping_OK : BOOL;
  G_Gateway_Data_Ready : BOOL;
  G_Gateway_Modbus_Registers : ARRAY[0..GVL_CONSTANTS.C_MAX_MODBUS_REGISTERS-1] OF WORD;
END_VAR

{attribute 'qualified_only'}
VAR_GLOBAL CONSTANT  (* GVL_CONSTANTS *)
  C_MAX_ZONES : INT := 16;  (* Максимальное количество зон (комнат) *)
  C_MAX_LIGHTING_ZONES : INT := 32;  (* Алиас для контуров освещения *)
  C_MAX_HEATING_CIRCUITS : INT := 8;  (* Алиас для контуров отопления *)
  C_MAX_CLIMATE_ZONES : INT := 16;  (* Алиас для климатических зон *)
  C_MAX_LIGHT_ZONES : INT := 32;  (* Алиас для световых зон *)
  C_MAX_SOCKETS : INT := 36;  (* Максимальное количество управляемых розеток *)
  C_MAX_BLINDS : INT := 20;  (* Максимальное количество штор/жалюзи *)
  C_MAX_ALARMS : INT := 20;  (* Максимальное количество активных тревог *)
  C_MAX_RULES : INT := 20;  (* Максимальное количество правил (движок правил) *)
  C_MAX_MANIFOLDS : INT := 5;  (* Максимальное количество коллекторов *)
  C_MAX_BOILERS : INT := 2;  (* Максимальное количество котлов *)
  C_MAX_SUPPLY_FANS : INT := 3;  (* Максимальное количество приточных вентиляторов *)
  C_MAX_EXHAUST_FANS : INT := 5;  (* Максимальное количество вытяжных вентиляторов *)
  C_MAX_SECURITY_SENSORS : INT := 15;  (* Максимальное количество датчиков безопасности (герконы, стекло) *)
  C_MAX_FLOOD_SENSORS : INT := 12;  (* Максимальное количество датчиков протечки *)
  C_MAX_DOOR_SENSORS : INT := 8;  (* Максимальное количество датчиков дверей *)
  C_MAX_CO_SENSORS : INT := 8;  (* Максимальное количество датчиков CO *)
  C_MAX_METHANE_SENSORS : INT := 2;  (* Максимальное количество датчиков метана *)
  C_MAX_VENT_UNITS : INT := 8;  (* Максимальное количество вентустановок *)
  C_MAX_SUPPLY_TEMPS : INT := 2;  (* Максимальное количество датчиков температуры притока *)
  C_MAX_SMOKE_SENSORS : INT := 6;  (* Максимальное количество датчиков дыма *)
  C_MAX_SCENARIOS : INT := 6;  (* Максимальное количество сценариев *)
  C_MAX_OUTDOOR_ZONES : INT := 4;  (* Максимальное количество зон уличного освещения *)
  C_MAX_ACCESS_CODES : INT := 10;  (* Максимальное количество кодов доступа *)
  C_MAX_WET_ZONES : INT := 4;  (* Максимальное количество "мокрых" зон (санузлы) *)
  C_MAX_CALIBRATIONS : INT := 20;  (* Максимальное количество калибровок датчиков *)
  C_MAX_MODULES : INT := 10;  (* Максимальное количество модулей ввода-вывода *)
  C_MAX_CLEANING_MODES : INT := 3;  (* Максимальное количество режимов уборки *)
  C_MAX_ALLOWED_IPS : INT := 5;  (* Максимальное количество разрешенных IP-адресов *)
  C_MAX_VENT_SUPPLY_MODES : INT := 3;  (* Максимальное количество режимов притока вентиляции *)
  C_MAX_SECURITY_PHONES : INT := 5;  (* Максимальное количество телефонов для оповещения *)
  C_MAX_FLOOD_VALVES : INT := 3;  (* Максимальное количество кранов защиты от протечек *)
  C_MAX_HUMIDITY_SENSORS : INT := 8;  (* Максимальное количество датчиков влажности *)
  C_MAX_CO2_SENSORS : INT := 8;  (* Максимальное количество датчиков CO2 *)
  C_MAX_CIRCUITS_PER_MANIFOLD : INT := 4;  (* Максимальное количество контуров на коллектор *)
  C_MAX_TREND_DATA_POINTS : INT := 100;  (* Максимальное количество точек данных для трендов *)
  C_MAX_HISTORY_RECORDS : INT := 100;  (* Максимальное количество записей в истории *)
  C_MAX_DEBUG_LOGS : INT := 1000;  (* Максимальное количество записей в логе отладки *)
  C_MAX_GATEWAY_COMMANDS : INT := 10;  (* Максимальное количество команд в буфере шлюза *)
  C_MAX_STATE_SNAPSHOTS : INT := 10;  (* Максимальное количество снимков состояния *)
  C_MAX_BLACKBOX_RECORDS : INT := 100;  (* Максимальное количество записей черного ящика *)
  C_MAX_PRESENCE_HISTORY : INT := 1008;  (* Максимальное количество записей истории присутствия *)
  C_MAX_MODBUS_REGISTERS : INT := 201;  (* Максимальное количество регистров Modbus *)
  C_MAX_DEDUPLICATION_HISTORY : INT := 100;  (* Максимальное количество записей истории дедупликации *)
  C_MAX_NVRAM_RECORDS : INT := 100;  (* Максимальное количество записей NVRAM *)
  C_MAX_NVRAM_DATA : INT := 128;  (* Максимальный размер данных NVRAM *)
  C_ANALOG_RAW_MAX : WORD := 27648;  (* Максимальное значение АЦП (100%) *)
  C_ANALOG_4MA_RAW : WORD := 5529;  (* Значение АЦП для 4mA (20% от 27648) *)
  C_ANALOG_3_6MA_RAW : WORD := 4976;  (* Порог обрыва NAMUR NE43 (< 3.6mA) *)
  C_ANALOG_21MA_RAW : WORD := 29030;  (* Порог КЗ NAMUR NE43 (> 21mA) *)
  C_ANALOG_10V_MAX_RAW : WORD := 30000;  (* Порог выхода за пределы 0-10V *)
  C_MS_IN_SECOND : UDINT := 1000;
  C_MS_IN_MINUTE : UDINT := 60000;
  C_MS_IN_HOUR : UDINT := 3600000;
  C_MS_IN_DAY : UDINT := 86400000;
  C_BOILER_CASCADE_MIN_DEMAND : REAL := 25.0;  (* Минимальный запрос для включения ведущего котла (5% от одного коллектора) *)
  C_BOILER_CASCADE_HIGH_DEMAND : REAL := 250.0;  (* Высокий запрос для включения второго котла (50% от общей мощности) *)
END_VAR

{attribute 'qualified_only'}
VAR_GLOBAL RETAIN  (* GVL_Retain *)
  G_Initialized : BOOL := FALSE;  (* Флаг инициализации retain-переменных *)
  G_NVRAM_Data : ARRAY[0..12799] OF BYTE;  (* 100 * 128 = 12800 байт *)
  G_BlackBox_Buffer : ARRAY[0..GVL_CONSTANTS.C_MAX_BLACKBOX_RECORDS-1] OF ST_BlackBox_Record;
  G_BlackBox_LastIndex : INT;
  G_BlackBox_Frozen : BOOL;
  G_Presence_History : ARRAY[0..GVL_CONSTANTS.C_MAX_PRESENCE_HISTORY-1] OF WORD;  (* 168 часов * 6 записей в час = 1008 записей (битовая маска 16 ламп) *)
  G_History_Buffer : ARRAY[1..GVL_CONSTANTS.C_MAX_HISTORY_RECORDS] OF ST_History_Record;
  G_History_Write_Idx : INT := 1;
  G_History_Total_Events : UDINT;
  G_Boiler_Accumulated_MS : ARRAY[1..GVL_CONSTANTS.C_MAX_BOILERS] OF UDINT;
  G_Boiler_Work_Seconds : ARRAY[1..GVL_CONSTANTS.C_MAX_BOILERS] OF UDINT;
  G_Valve_Test_Results : ARRAY[1..GVL_CONSTANTS.C_MAX_MANIFOLDS] OF BOOL;
  G_Access_Codes : ARRAY[1..GVL_CONSTANTS.C_MAX_ACCESS_CODES] OF DWORD := [16#9BE3E0A3, 16#4A89A12D, 16#F4DBDF21, 16#90F59C65, 16#0972D346, 0, 0, 0, 0, 0];
  G_RFID_Tags : ARRAY[1..GVL_CONSTANTS.C_MAX_ACCESS_CODES] OF STRING(20) := ['A1B2C3D4', 'E5F67890', '', '', '', '', '', '', '', ''];
END_VAR

{attribute 'qualified_only'}
VAR_GLOBAL  (* GVL_HEALTH_BRIDGE *)
  G_Smoke_Detected : BOOL;
  G_Gas_Detected : BOOL;
  G_Leak_Detected : BOOL;
  G_Leak_Warning_Level : BOOL;
  G_CO_Warning_Level : BOOL;
  G_CO_Alarm_Level : BOOL;
  G_Last_Fault_Event_Text : STRING(255);
END_VAR

{attribute 'qualified_only'}
VAR_GLOBAL  (* GVL_COMMAND *)
  G_Gas_Valve_Close : BOOL := FALSE;  (* Команда: Закрыть газовый клапан *)
  G_Boiler_Stop : BOOL := FALSE;  (* Команда: Остановка котлов *)
  G_Supply_100_Req : BOOL := FALSE;  (* Команда: Приток 100% *)
  G_Supply_80_Req : BOOL := FALSE;  (* Команда: Приток 80% *)
  G_Vent_PV3_Boost : BOOL := FALSE;  (* Команда: Форсированный режим ПВ-3 *)
  G_Exhaust_100_Req : BOOL := FALSE;  (* Команда: Вытяжка 100% *)
  G_Vent_Stop : BOOL := FALSE;  (* Команда: Остановка вентиляции *)
  G_Close_Valve_35 : BOOL := FALSE;  (* Команда: Закрыть вводной кран 1 *)
  G_Close_Valve_36 : BOOL := FALSE;  (* Команда: Закрыть вводной кран 2 *)
  G_Gate_Open : BOOL;
  G_Wicket_Open : BOOL;
  G_Lock_1_Open : BOOL;
  G_Lock_1_Close : BOOL;
  G_Lock_2_Open : BOOL;
  G_Lock_2_Close : BOOL;
  G_Reset_Errors : BOOL := FALSE;  (* Команда: Сброс ошибок *)
  G_Scenario_Request : E_SCENARIO_TYPE := E_SCENARIO_TYPE.SCENARIO_NONE;  (* Запрос на активацию сценария *)
  G_Arm_Req : BOOL;
  G_Disarm_Req : BOOL;
  G_PIN_Code : STRING(4);
  G_RFID_Tag : STRING(20);
  G_2FA_Code_In : STRING(6);
  G_Send_2FA_Req : BOOL;
  G_2FA_Code_Out : STRING(6);
  G_Lighting_Override : ARRAY[1..32] OF BYTE;
  G_Blinds_Override : ARRAY[1..GVL_CONSTANTS.C_MAX_BLINDS] OF BYTE;
  G_Socket_Override : ARRAY[1..GVL_CONSTANTS.C_MAX_SOCKETS] OF BOOL;
  CMD_Set_Manifold_Pump_In_Service : ARRAY[1..GVL_CONSTANTS.C_MAX_MANIFOLDS] OF BOOL;
  CMD_Set_DHW_Heating_Pump_In_Service : BOOL;
  CMD_Set_DHW_Circ_Pump_In_Service : BOOL;
  CMD_Dangerous_Action_Confirm : BOOL;
  CMD_Dangerous_Action_Request : BOOL;
  CMD_User_Access_Level : INT := 0;
  CMD_Valve_Test_Open : BOOL;
  CMD_Valve_Test_Close : BOOL;
  CMD_Valve_Test_Confirm : BOOL;
  CMD_Water_Valve_Test_Open : BOOL;
  CMD_Water_Valve_Test_Close : BOOL;
  CMD_Water_Valve_Test_Confirm : BOOL;
  CMD_Gas_Valve_Test_Open : BOOL;
  CMD_Gas_Valve_Test_Close : BOOL;
  CMD_Gas_Valve_Test_Confirm : BOOL;
  CMD_Water_Selective_Recover : BOOL;
  CMD_Gas_Selective_Recover : BOOL;
END_VAR

{attribute 'qualified_only'}
VAR_GLOBAL  (* GVL_ALARM *)
  G_Security_Armed : BOOL := FALSE;  (* Флаг: Система безопасности активирована *)
  G_Security_Siren : BOOL := FALSE;
  G_Global_Siren : BOOL := FALSE;  (* Глобальный флаг сирены от Alarm Manager *)
  G_Global_Critical : BOOL := FALSE;
  G_Global_Warning : BOOL := FALSE;
  G_Active_Alarm_Count : INT := 0;
  G_Unacked_Alarm_Count : INT := 0;
  G_Alarm_List : ARRAY[1..GVL_CONSTANTS.C_MAX_ALARMS] OF ST_Alarm_Record;
  G_Gas_Alarm_Active : BOOL := FALSE;  (* Флаг: Обнаружена критическая концентрация газа *)
  G_Gas_Fire_Siren : BOOL := FALSE;
  G_Fire_Alarm_Active : BOOL := FALSE;  (* Флаг: Сработали пожарные датчики *)
  G_Flood_Alarm_Active : BOOL := FALSE;  (* Флаг: Обнаружена протечка воды *)
  G_Security_Alarm : BOOL := FALSE;  (* Флаг: Тревога системы безопасности *)
END_VAR

{attribute 'qualified_only'}
VAR_GLOBAL  (* GVL_STATE *)
  G_Floor_Temps : ARRAY[1..8] OF REAL;  (* Массив текущих температур поверхности пола *)
  G_Room_Temps : ARRAY[1..GVL_CONSTANTS.C_MAX_ZONES] OF REAL;
  G_Room_Hum : ARRAY[1..GVL_CONSTANTS.C_MAX_ZONES] OF REAL;
  G_Room_CO2 : ARRAY[1..GVL_CONSTANTS.C_MAX_ZONES] OF REAL;
  G_Motion_Sensors : ARRAY[1..32] OF BOOL;
  G_Door_Sensors : ARRAY[1..GVL_CONSTANTS.C_MAX_DOOR_SENSORS] OF BOOL;
  G_Window_Sensors : ARRAY[1..GVL_CONSTANTS.C_MAX_ZONES] OF BOOL;
  G_Water_Sensors : ARRAY[1..GVL_CONSTANTS.C_MAX_FLOOD_SENSORS] OF BOOL;
  G_Smoke_Sensors : ARRAY[1..GVL_CONSTANTS.C_MAX_SMOKE_SENSORS] OF BOOL;
  G_Methane_Sensors : ARRAY[1..GVL_CONSTANTS.C_MAX_METHANE_SENSORS] OF REAL;
  G_CO_Sensors : ARRAY[1..GVL_CONSTANTS.C_MAX_CO_SENSORS] OF REAL;
  G_Manifold_Pressures : ARRAY[1..GVL_CONSTANTS.C_MAX_MANIFOLDS] OF REAL;
  G_Manifold_Currents : ARRAY[1..GVL_CONSTANTS.C_MAX_MANIFOLDS] OF REAL;
  G_Manifold_T_Supply : ARRAY[1..GVL_CONSTANTS.C_MAX_MANIFOLDS] OF REAL;
  G_Manifold_T_Return : ARRAY[1..GVL_CONSTANTS.C_MAX_MANIFOLDS] OF REAL;
  G_Boiler_Flame : ARRAY[1..GVL_CONSTANTS.C_MAX_BOILERS] OF BOOL;
  G_Boiler_Error : ARRAY[1..GVL_CONSTANTS.C_MAX_BOILERS] OF BOOL;
  G_Boiler_OT_Online : ARRAY[1..GVL_CONSTANTS.C_MAX_BOILERS] OF BOOL;  (* Статус доступности OpenTherm-канала котла от реального OT-адаптера/драйвера *)
  G_Boiler_OT_Enable : ARRAY[1..GVL_CONSTANTS.C_MAX_BOILERS] OF BOOL;  (* Команды разрешения через OpenTherm *)
  G_Boiler_OT_Setpoint : ARRAY[1..GVL_CONSTANTS.C_MAX_BOILERS] OF REAL;  (* Уставки через OpenTherm *)
  G_Physical_Switches : ARRAY[1..32] OF BOOL;
  G_Socket_Switches : ARRAY[1..GVL_CONSTANTS.C_MAX_SOCKETS] OF BOOL;  (* Legacy-поле: локальные выключатели розеток не используются *)
  G_Outdoor_Temp : REAL;
  G_Supply_Temps : ARRAY[1..GVL_CONSTANTS.C_MAX_SUPPLY_TEMPS] OF REAL;  (* Температура приточного воздуха после калорифера *)
  G_DHW_Temp : REAL;
  G_DHW_Pressure : REAL;
  G_Zone_Valves : ARRAY[1..8] OF BOOL;
  G_Manifold_Pumps : ARRAY[1..GVL_CONSTANTS.C_MAX_MANIFOLDS] OF BOOL;
  G_Manifold_Valves : ARRAY[1..GVL_CONSTANTS.C_MAX_MANIFOLDS] OF REAL;  (* 0.0 - 1.0 *)
  G_Manifold_End_Switches : ARRAY[1..GVL_CONSTANTS.C_MAX_MANIFOLDS] OF BOOL;  (* Концевики клапанов *)
  G_Supply_Fans : ARRAY[1..GVL_CONSTANTS.C_MAX_SUPPLY_FANS] OF REAL;  (* 0.0 - 1.0 *)
  G_Exhaust_Fans : ARRAY[1..GVL_CONSTANTS.C_MAX_EXHAUST_FANS] OF REAL;  (* 0.0 - 1.0 *)
  G_Vent_Heater_Power : ARRAY[1..GVL_CONSTANTS.C_MAX_BOILERS] OF REAL;
  G_Lighting_Levels : ARRAY[1..32] OF BYTE;
  G_Blinds_Positions : ARRAY[1..GVL_CONSTANTS.C_MAX_BLINDS] OF BYTE;
  G_Socket_States : ARRAY[1..GVL_CONSTANTS.C_MAX_SOCKETS] OF BOOL;
  G_DHW_Heating_Pump : BOOL;
  G_DHW_Circ_Pump : BOOL;
  G_Backup_Circulation_Pump : BOOL;  (* Резервный циркуляционный насос для антизамерзания при газовой аварии *)
  G_Electric_Heater_Enable : BOOL;  (* Сухой контакт электрического нагревателя для антизамерзания *)
  G_Safety_Gas_Alarm : BOOL;
  G_Safety_Leak_Alarm : BOOL;
  G_Safety_Smoke_Alarm : BOOL;
  G_Safety_Emergency_Stop : BOOL;  (* агрегированный аварийный стоп *)
  G_Safety_Gas_Latched : BOOL;  (* защёлкнутая газовая авария *)
  G_Safety_Leak_Latched : BOOL;  (* защёлкнутая авария протечки *)
  G_Safety_Smoke_Latched : BOOL;  (* защёлкнутая дымовая/пожарная авария *)
  G_Safety_Freeze_Risk : BOOL;  (* риск замерзания при защёлкнутой газовой аварии *)
  G_System_Mode : E_System_Operating_Mode := E_System_Operating_Mode.MODE_NORMAL;  (* Текущий режим работы системы *)
  G_System_Mode_Text : STRING(64);
  G_Heating_IO_Fault : BOOL;
  G_Heating_Sensor_Fault : BOOL;
  G_Heating_Subsystem_Degraded : BOOL;
  G_DHW_IO_Fault : BOOL;
  G_DHW_Sensor_Fault : BOOL;
  G_DHW_Subsystem_Degraded : BOOL;
  G_Ventilation_IO_Fault : BOOL;
  G_Ventilation_Subsystem_Degraded : BOOL;
  G_Lighting_IO_Fault : BOOL;
  G_Lighting_Subsystem_Degraded : BOOL;
  G_Access_Comm_Fault : BOOL;
  G_Evacuation_Lighting_Active : BOOL;
  G_Evac_Hazard_Zone : ARRAY[1..32] OF BOOL;  (* опасные зоны (дым/протечка) *)
  G_Evac_Guidance : ARRAY[1..32] OF INT;  (* -1 = избегать, 0 = нейтрально, +1 = к выходу *)
  G_Rule_Actions : ARRAY[1..GVL_CONSTANTS.C_MAX_RULES] OF ST_Rule_Action;
  G_Sim_Lights : ARRAY[1..32] OF BOOL;
  G_Freeze_Hardware_Degraded : BOOL;  (* Деградация anti-freeze hardware *)
  G_Freeze_Hardware_Failed : BOOL;  (* Критический отказ anti-freeze hardware *)
  G_Water_Zone_Enable : ARRAY[1..32] OF BOOL;  (* Селективное открытие воды по зонам *)
  G_Water_Zone_Open_FB : ARRAY[1..32] OF BOOL;  (* Обратная связь: зональный клапан открыт *)
  G_Water_Zone_Close_FB : ARRAY[1..32] OF BOOL;  (* Обратная связь: зональный клапан закрыт *)
  G_Water_Zone_Exercise_Active : ARRAY[1..32] OF BOOL;  (* Профилактическая прокрутка шаровых кранов *)
END_VAR

{attribute 'qualified_only'}
VAR_GLOBAL  (* GVL_DEBUG *)
  G_Device_Health_Zones : ARRAY[1..GVL_CONSTANTS.C_MAX_CLIMATE_ZONES] OF ST_Device_Health;
  G_Device_Health_Manifolds : ARRAY[1..GVL_CONSTANTS.C_MAX_MANIFOLDS] OF ST_Device_Health;
  G_Device_Health_Boilers : ARRAY[1..GVL_CONSTANTS.C_MAX_BOILERS] OF ST_Device_Health;
  G_Device_Health_Vents : ARRAY[1..GVL_CONSTANTS.C_MAX_MANIFOLDS] OF ST_Device_Health;
  G_System_Health_Summary : BYTE := 100;
  G_Pump_Health : ARRAY[1..GVL_CONSTANTS.C_MAX_MANIFOLDS] OF ST_Device_Health;  (* Для 5 коллекторных насосов *)
  G_Gas_Valve_Health : ST_Device_Health;
END_VAR

{attribute 'qualified_only'}
VAR_GLOBAL  (* GVL_IO *)
  DI_Security_Open : ARRAY[1..GVL_CONSTANTS.C_MAX_SECURITY_SENSORS] OF BOOL;  (* Дискретные входы: Герконы (нормально-замкнутые контакты, TRUE = Открыто) *)
  DI_Security_Glass : ARRAY[1..GVL_CONSTANTS.C_MAX_SECURITY_SENSORS] OF BOOL;  (* Дискретные входы: Датчики разбития стекла (активный уровень - TRUE) *)
  DI_Security_2F_Group : BOOL;  (* Дискретный вход: Групповой шлейф безопасности 2-го этажа (общий сигнал) *)
  DI_Flood_Sensors : ARRAY[1..GVL_CONSTANTS.C_MAX_FLOOD_SENSORS] OF BOOL;  (* Дискретные входы: Датчики протечки воды (активный уровень - TRUE) *)
  DI_Manifold_End_Switches : ARRAY[1..GVL_CONSTANTS.C_MAX_MANIFOLDS] OF BOOL;  (* Дискретные входы: Концевые выключатели клапанов коллекторов *)
  AO_Manifold_Valves : ARRAY[1..GVL_CONSTANTS.C_MAX_MANIFOLDS] OF UINT;  (* Аналоговые выходы: Приводы клапанов (0-10В, 0-1000 ед. для Modbus) *)
  DO_Manifold_Pumps : ARRAY[1..GVL_CONSTANTS.C_MAX_MANIFOLDS] OF BOOL;  (* Дискретные выходы: Циркуляционные насосы коллекторных узлов (220В) *)
  AI_Manifold_Currents : ARRAY[1..GVL_CONSTANTS.C_MAX_MANIFOLDS] OF INT;  (* Аналоговые входы: Обратная связь по току потребления насосов (диагностика) *)
  AI_Manifold_Pressures : ARRAY[1..GVL_CONSTANTS.C_MAX_MANIFOLDS] OF INT;  (* Аналоговые входы: Давление теплоносителя в коллекторах (0-10 бар) *)
  AI_Manifold_Temps_Supply : ARRAY[1..GVL_CONSTANTS.C_MAX_MANIFOLDS] OF ST_Owen_Analog_Value;  (* Аналоговые входы: Температура подачи (структура со статусом) *)
  AI_Manifold_Temps_Return : ARRAY[1..GVL_CONSTANTS.C_MAX_MANIFOLDS] OF INT;  (* Аналоговые входы: Температура обратной линии (в 10-х долях градуса) *)
  AO_Supply_Fans : ARRAY[1..GVL_CONSTANTS.C_MAX_SUPPLY_FANS] OF UINT;  (* Аналоговые выходы: Скорость приточных вентиляторов (0-10В) *)
  AO_Exhaust_Fans : ARRAY[1..GVL_CONSTANTS.C_MAX_EXHAUST_FANS] OF UINT;  (* Аналоговые выходы: Скорость вытяжных вентиляторов (0-10В) *)
  AO_Lighting_Levels : ARRAY[1..GVL_CONSTANTS.C_MAX_ZONES] OF UINT;  (* Аналоговые выходы: диммирование освещения (0-1000 -> 0..100%) *)
  AO_Blinds_Positions : ARRAY[1..GVL_CONSTANTS.C_MAX_BLINDS] OF UINT;  (* Аналоговые выходы: позиционирование штор/жалюзи (0-1000 -> 0..100%) *)
  AI_Supply_Temps : ARRAY[1..GVL_CONSTANTS.C_MAX_SUPPLY_TEMPS] OF ST_Owen_Analog_Value;  (* Аналоговые входы: Температура приточного воздуха после калорифера *)
  AI_Boiler_Modulation : ARRAY[1..GVL_CONSTANTS.C_MAX_BOILERS] OF INT;  (* Аналоговые входы: Текущий уровень модуляции мощности котла (%) *)
  AI_Boiler_Flame_Status : ARRAY[1..GVL_CONSTANTS.C_MAX_BOILERS] OF BOOL;  (* Дискретные входы: Датчик ионизации (подтверждение наличия пламени) *)
  DI_Boiler_Error : ARRAY[1..GVL_CONSTANTS.C_MAX_BOILERS] OF BOOL;  (* Дискретные входы: Сигнал общей ошибки/аварии котла *)
  AI_Methane_LEL : ARRAY[1..GVL_CONSTANTS.C_MAX_METHANE_SENSORS] OF ST_Owen_Analog_Value;  (* Аналоговые входы: Уровень метана CH4 (0-100% LEL) *)
  AI_CO_PPM : ARRAY[1..GVL_CONSTANTS.C_MAX_CO_SENSORS] OF REAL;  (* Аналоговые входы: Уровень угарного газа CO (PPM) *)
  DI_Smoke_Sensors : ARRAY[1..GVL_CONSTANTS.C_MAX_SMOKE_SENSORS] OF BOOL;  (* Дискретные входы: Оптические датчики дыма (пожарный шлейф) *)
  AI_Temp_Outdoor : ST_Owen_Analog_Value;  (* Аналоговый вход: Наружная температура воздуха (уличный датчик) *)
  AI_Floor_Temps : ARRAY[1..GVL_CONSTANTS.C_MAX_ZONES] OF REAL;  (* Аналоговые входы: Температура стяжки пола по зонам (датчики в гильзах) *)
  AI_Room_Temps : ARRAY[1..GVL_CONSTANTS.C_MAX_ZONES] OF REAL;  (* Аналоговые входы: Температура воздуха в помещениях (настенные датчики) *)
  AI_Room_Hum : ARRAY[1..GVL_CONSTANTS.C_MAX_ZONES] OF REAL;  (* Аналоговые входы: Влажность воздуха в помещениях (%) *)
  AI_Room_CO2 : ARRAY[1..GVL_CONSTANTS.C_MAX_ZONES] OF REAL;  (* Аналоговые входы: Уровень CO2 в помещениях (ppm) *)
  DO_Zone_Valves : ARRAY[1..GVL_CONSTANTS.C_MAX_ZONES] OF BOOL;  (* Дискретные выходы: Термоэлектрические приводы контуров (220В) *)
  AI_DHW_Temp : REAL;  (* Аналоговый вход: Температура воды в бойлере косвенного нагрева *)
  AI_DHW_Pressure : REAL;  (* Аналоговый вход: Давление в контуре ГВС (контроль подпитки и утечек) *)
  DO_DHW_Heating_Pump : BOOL;  (* Дискретный выход: Насос загрузки бойлера (первичный контур от котла) *)
  DO_DHW_Circ_Pump : BOOL;  (* Дискретный выход: Насос рециркуляции ГВС (кольцо потребителей) *)
  DO_Backup_Circulation_Pump : BOOL;  (* Дискретный выход: Резервный циркуляционный насос антизамерзания *)
  DO_Electric_Heater_Enable : BOOL;  (* Дискретный выход: Сухой контакт электрического нагревателя антизамерзания *)
  DI_Lighting_Switches : ARRAY[1..GVL_CONSTANTS.C_MAX_ZONES] OF BOOL;  (* Дискретные входы: Физические кнопки/выключатели (импульсные) *)
  DI_Socket_Switches : ARRAY[1..GVL_CONSTANTS.C_MAX_SOCKETS] OF BOOL;  (* Legacy-вход: локальные выключатели розеток отключены концептуально *)
  DI_Motion_Sensors : ARRAY[1..GVL_CONSTANTS.C_MAX_ZONES] OF BOOL;  (* Дискретные входы: Датчики присутствия (PIR-сенсоры) *)
  DO_Sockets : ARRAY[1..GVL_CONSTANTS.C_MAX_SOCKETS] OF BOOL;  (* Дискретные выходы: Управление розетками (реле) *)
  DO_Gas_Valve_Close : BOOL;  (* Дискретный выход: Импульс на закрытие электромагнитного газового клапана *)
  DO_Water_Valve_35_Close : BOOL;  (* Дискретный выход: Закрыть вводной шаровый кран воды №1 (с электроприводом) *)
  DO_Water_Valve_36_Close : BOOL;  (* Дискретный выход: Закрыть вводной шаровый кран воды №2 (с электроприводом) *)
  AI_Water_Valve_35_Current : REAL;  (* Аналоговый вход: Ток потребления электропривода крана №1 (контроль заклинивания) *)
  AI_Water_Valve_36_Current : REAL;  (* Аналоговый вход: Ток потребления электропривода крана №2 (контроль заклинивания) *)
  DI_Power_OK : BOOL;  (* Дискретный вход: Контроль наличия напряжения на вводе (реле контроля фаз) *)
  DO_Gas_Siren : BOOL;  (* Дискретный выход: Звуковое оповещение при опасной концентрации газа *)
  DO_Fire_Siren : BOOL;  (* Дискретный выход: Звуковое оповещение при обнаружении задымления *)
  DO_Security_Siren : BOOL;  (* Дискретный выход: Сирена охранной сигнализации *)
  DO_Pump_Main_Enable : BOOL;  (* Дискретный выход: Разрешение работы главного циркуляционного насоса системы *)
  DO_Gate_Open : BOOL;  (* Дискретный выход: Команда на открытие въездных ворот (импульс) *)
  DO_Wicket_Open : BOOL;  (* Дискретный выход: Команда на разблокировку электрозамка калитки *)
  DO_Lock_1_Open : BOOL;  (* Дискретный выход: Разблокировать основной электромеханический замок дома *)
  DO_Lock_1_Close : BOOL;  (* Дискретный выход: Заблокировать основной электромеханический замок дома *)
  DO_Lock_2_Open : BOOL;  (* Дискретный выход: Разблокировать дополнительный замок (черный ход) *)
  DO_Lock_2_Close : BOOL;  (* Дискретный выход: Заблокировать дополнительный замок (черный ход) *)
  DI_Partner_Pulse : BOOL;  (* Дискретный вход: Пульс от второго ПЛК *)
  DI_Partner_Active : BOOL;  (* Дискретный вход: Статус активности второго ПЛК *)
  DO_Heartbeat_Pulse : BOOL;  (* Дискретный выход: Собственный пульс *)
  DO_Active_Status : BOOL;  (* Дискретный выход: Собственный статус активности *)
  DI_Module_1_Heartbeat : BOOL;  (* Сигнал жизни от модуля 1 *)
  DI_Module_2_Heartbeat : BOOL;  (* Сигнал жизни от модуля 2 *)
  DI_Backup_Circulation_Pump_Feedback : BOOL;  (* Обратная связь резервного циркуляционного насоса *)
  DI_Electric_Heater_Feedback : BOOL;  (* Обратная связь электрического нагревателя *)
  DI_Water_Zone_Open_FB : ARRAY[1..32] OF BOOL;  (* Концевики: зональный водяной клапан открыт *)
  DI_Water_Zone_Close_FB : ARRAY[1..32] OF BOOL;  (* Концевики: зональный водяной клапан закрыт *)
  DO_Water_Zone_Enable : ARRAY[1..32] OF BOOL;  (* Разрешение подачи воды по зонам *)
END_VAR

{attribute 'qualified_only'}
VAR_GLOBAL  (* GVL_STATUS *)
  G_System_Time_MS : UDINT;  (* Системное время в миллисекундах *)
  G_Last_System_Time_MS : UDINT := 0;  (* Предыдущее системное время (для детекции переполнения) *)
  G_Time_Of_Day_MS : UDINT := 0;  (* Время от начала суток в мс (0-86399999) *)
  G_Current_Day : UINT := 1;  (* Текущий день недели (1-7) *)
  G_Day_Of_Year : UINT := 1;  (* Текущий день года (1-365) *)
  G_Current_TOD : TOD;  (* Текущее время суток *)
  G_Current_Scenario : E_SCENARIO_TYPE := E_SCENARIO_TYPE.SCENARIO_NONE;  (* Текущий активный сценарий *)
  G_Previous_Scenario : E_SCENARIO_TYPE := E_SCENARIO_TYPE.SCENARIO_NONE;  (* Предыдущий сценарий *)
  G_Is_Night : BOOL;  (* Флаг ночного времени *)
  G_PLC_ID : BYTE := 1;  (* 1 = PLC_A, 2 = PLC_B *)
  G_Is_Active_PLC : BOOL;
  G_Local_PLC_ID : BYTE := 1;  (* Идентификатор данного ПЛК в паре *)
  G_Active_PLC_ID : BYTE := 1;  (* Идентификатор ведущего ПЛК *)
  G_Remote_PLC_Pulse : BOOL;  (* Сигнал "жизни" от второго ПЛК *)
  G_Security_Status_Msg : STRING(200);
  G_Gas_Status_Msg : STRING(200);
  G_Flood_Status_Msg : STRING(200);
  G_Vent_Status_Msg : STRING(200);
  G_DHW_Status : ST_DHW_Status;
  G_Manifold_Status : ARRAY[1..GVL_CONSTANTS.C_MAX_MANIFOLDS] OF ST_Manifold_Status;
  G_Boiler_Status : ARRAY[1..GVL_CONSTANTS.C_MAX_BOILERS] OF ST_Boiler_Status;
  G_IO_Modules_Online : ARRAY[1..GVL_CONSTANTS.C_MAX_MODULES] OF BOOL;  (* Статусы модулей ввода-вывода *)
  G_Sim_Active : BOOL;
  G_Wet_Zone_Light_Active : BOOL;
  G_System_Mode_Msg : STRING(200);  (* Пояснение текущего режима работы системы для HMI *)
  G_System_Mode_Cause : STRING(200);  (* Корневая причина режима (пожар/газ/протечка/штатно) *)
  G_Evac_Target_Zone_Name : STRING(80);  (* Предпочтительная зона выхода/направления эвакуации *)
  G_Evac_Hazard_Zone_Name : STRING(80);  (* Наиболее важная опасная зона для HMI/диагностики *)
  G_Diagnostics : ST_System_Diagnostics;  (* Интегральная диагностика и HMI-состояния *)
END_VAR

FUNCTION_BLOCK FB_Rule_Compatibility_Package
  VAR_INPUT
    VI_Rule_Legacy : ST_User_Rule;
  END_VAR
  VAR_OUTPUT
    VO_Forward_OK : BOOL;
    VO_Reverse_OK : BOOL;
    VO_Warning_Text : STRING(255);
    VO_Rule_Legacy_Roundtrip : ST_Rule;
  END_VAR

            VO_Forward_OK := TRUE;
VO_Reverse_OK := TRUE;
VO_Warning_Text := '';

VO_Rule_Legacy_Roundtrip.Action_Type := VI_Rule_Legacy.Action_Type;
VO_Rule_Legacy_Roundtrip.Action_Target_ID := VI_Rule_Legacy.Action_Target_ID;
VO_Rule_Legacy_Roundtrip.Action_Value := VI_Rule_Legacy.Action_Value;
VO_Rule_Legacy_Roundtrip.Condition_Type := VI_Rule_Legacy.Condition_Type;
VO_Rule_Legacy_Roundtrip.Condition_Target_ID := VI_Rule_Legacy.Condition_Target_ID;
VO_Rule_Legacy_Roundtrip.Condition_Op := VI_Rule_Legacy.Condition_Op;
VO_Rule_Legacy_Roundtrip.Condition_Value := VI_Rule_Legacy.Condition_Value;
VO_Rule_Legacy_Roundtrip.Condition_Value_Max := VI_Rule_Legacy.Condition_Value_Max;
          
END_FUNCTION_BLOCK

FUNCTION_BLOCK FB_Lifetime_Predictor
  VAR_INPUT
    VI_Runtime_Hours : UDINT;
    VI_Start_Count : UDINT;
    VI_Nominal_Life : UDINT := 10000;
  END_VAR
  VAR_OUTPUT
    VO_Remaining_Percent : BYTE;
    VO_Maintenance_Req : BOOL;
  END_VAR

            // Упрощенная модель износа
IF VI_Nominal_Life > 0 THEN
    VO_Remaining_Percent := TO_BYTE(100 - (VI_Runtime_Hours * 100 / VI_Nominal_Life));
ELSE
    VO_Remaining_Percent := 0;
END_IF;

VO_Maintenance_Req := (VO_Remaining_Percent < 10);
          
END_FUNCTION_BLOCK

FUNCTION_BLOCK FB_Manifold_Pump_Controller
  VAR_INPUT
    VI_Enable_Request : BOOL;
    VI_System_Time : UDINT;
    VI_Stop_Ramp_MS : UDINT := 5000;
  END_VAR
  VAR_OUTPUT
    VO_Speed_Percent : BYTE;
    VO_Running : BOOL;
  END_VAR
  VAR
    L_Stop_Start_Time : UDINT;
    L_Stopping : BOOL;
    L_elapsed : UDINT;
  END_VAR

            IF VI_Enable_Request THEN
    VO_Speed_Percent := 100;
    VO_Running := TRUE;
    L_Stopping := FALSE;
ELSE
    IF VO_Running AND NOT L_Stopping THEN
        L_Stopping := TRUE;
        L_Stop_Start_Time := VI_System_Time;
    END_IF;
    
    IF L_Stopping THEN
        L_elapsed := (SEL(VI_System_Time >= L_Stop_Start_Time, VI_System_Time - L_Stop_Start_Time, (4294967295 - L_Stop_Start_Time) + VI_System_Time + 1));
        IF L_elapsed < VI_Stop_Ramp_MS THEN
            // Исправлено: защита от отрицательного значения
            VO_Speed_Percent := REAL_TO_BYTE(100.0 * (1.0 - TO_REAL(L_elapsed) / TO_REAL(VI_Stop_Ramp_MS)));
        ELSE
            VO_Speed_Percent := 0;
            VO_Running := FALSE;
            L_Stopping := FALSE;
        END_IF;
    END_IF;
END_IF;
          
END_FUNCTION_BLOCK

FUNCTION_BLOCK FB_Boiler_Cascade_Manager
  VAR_INPUT
    VI_Enable : BOOL;
    VI_System_Time_MS : UDINT;
    VI_Boiler_Stop : BOOL;
    VI_DHW_Heating_Demand : BOOL;
    VI_DHW_Target_Temp : REAL;
    VI_Target_Supply_Temp : REAL;
    VI_Demand_Power : REAL;
    VI_Boiler_Flame_Status : ARRAY[1..GVL_CONSTANTS.C_MAX_BOILERS] OF BOOL;
    VI_Boiler_Error_Status : ARRAY[1..GVL_CONSTANTS.C_MAX_BOILERS] OF BOOL;
    VI_Boiler_OT_Online : ARRAY[1..GVL_CONSTANTS.C_MAX_BOILERS] OF BOOL;
    VI_Boiler_Modulation : ARRAY[1..GVL_CONSTANTS.C_MAX_BOILERS] OF REAL;
  END_VAR
  VAR_OUTPUT
    VO_Boiler_Enable : ARRAY[1..GVL_CONSTANTS.C_MAX_BOILERS] OF BOOL;
    VO_Boiler_Setpoint : ARRAY[1..GVL_CONSTANTS.C_MAX_BOILERS] OF REAL;
    VO_Lead_Boiler : BYTE;
  END_VAR
  VAR
    L_i : INT;
    L_Lead_Boiler : BYTE := 1;
    L_Last_Rotation_MS : UDINT := 0;
    L_Rotation_Initialized : BOOL := FALSE;
    L_Rotation_Period_MS : UDINT := 604800000;
    L_Lead_Available : BOOL;
    L_Reserve_Available : BOOL;
    L_Reserve_Boiler : BYTE;
    L_Start_Reserve : BOOL;
    L_Target_Setpoint : REAL;
    L_Flame_Miss_Timer : ARRAY[1..GVL_CONSTANTS.C_MAX_BOILERS] OF TON;
  END_VAR

            // Сброс выходов по умолчанию
FOR L_i := 1 TO GVL_CONSTANTS.C_MAX_BOILERS DO
    VO_Boiler_Enable[L_i] := FALSE;
    VO_Boiler_Setpoint[L_i] := 0.0;
END_FOR;

// Инициализация ротации
IF NOT L_Rotation_Initialized THEN
    L_Last_Rotation_MS := VI_System_Time_MS;
    L_Rotation_Initialized := TRUE;
END_IF;

// Принудительная остановка
IF VI_Boiler_Stop THEN
    VO_Lead_Boiler := L_Lead_Boiler;
    RETURN;
END_IF;

// Ротация строго каждые 168 часов
IF (VI_System_Time_MS - L_Last_Rotation_MS) >= L_Rotation_Period_MS THEN
    IF GVL_CONSTANTS.C_MAX_BOILERS > 1 THEN
        L_Lead_Boiler := 3 - L_Lead_Boiler;
    END_IF;
    L_Last_Rotation_MS := VI_System_Time_MS;
END_IF;

L_Reserve_Boiler := SEL(L_Lead_Boiler = 1, 1, 2);

L_Lead_Available :=
    VI_Boiler_OT_Online[L_Lead_Boiler] AND
    NOT VI_Boiler_Error_Status[L_Lead_Boiler];

L_Reserve_Available :=
    (GVL_CONSTANTS.C_MAX_BOILERS > 1) AND
    VI_Boiler_OT_Online[L_Reserve_Boiler] AND
    NOT VI_Boiler_Error_Status[L_Reserve_Boiler];

// Контроль "команда есть, пламени нет" для ведущего котла
L_Flame_Miss_Timer[L_Lead_Boiler](
    IN := VI_Enable AND L_Lead_Available AND NOT VI_DHW_Heating_Demand AND NOT VI_Boiler_Flame_Status[L_Lead_Boiler],
    PT := T#120s
);

IF L_Flame_Miss_Timer[L_Lead_Boiler].Q AND L_Reserve_Available THEN
    L_Lead_Boiler := L_Reserve_Boiler;
    L_Last_Rotation_MS := VI_System_Time_MS;
    L_Lead_Available :=
        VI_Boiler_OT_Online[L_Lead_Boiler] AND
        NOT VI_Boiler_Error_Status[L_Lead_Boiler];
    L_Reserve_Boiler := SEL(L_Lead_Boiler = 1, 1, 2);
    L_Reserve_Available :=
        (GVL_CONSTANTS.C_MAX_BOILERS > 1) AND
        VI_Boiler_OT_Online[L_Reserve_Boiler] AND
        NOT VI_Boiler_Error_Status[L_Reserve_Boiler];
END_IF;

// Нет запроса тепла
IF NOT VI_Enable THEN
    VO_Lead_Boiler := L_Lead_Boiler;
    RETURN;
END_IF;

// Целевая уставка
IF VI_DHW_Heating_Demand THEN
    L_Target_Setpoint := LIMIT(20.0, VI_DHW_Target_Temp + 15.0, 85.0);
ELSE
    L_Target_Setpoint := LIMIT(20.0, VI_Target_Supply_Temp + 5.0, 80.0);
END_IF;

// Выбор ведущего по доступности
IF NOT L_Lead_Available AND L_Reserve_Available THEN
    L_Lead_Boiler := L_Reserve_Boiler;
    L_Lead_Available := TRUE;
    L_Reserve_Boiler := SEL(L_Lead_Boiler = 1, 1, 2);
    L_Reserve_Available :=
        (GVL_CONSTANTS.C_MAX_BOILERS > 1) AND
        VI_Boiler_OT_Online[L_Reserve_Boiler] AND
        NOT VI_Boiler_Error_Status[L_Reserve_Boiler];
END_IF;

// Основной котёл
IF L_Lead_Available THEN
    VO_Boiler_Enable[L_Lead_Boiler] := TRUE;
    VO_Boiler_Setpoint[L_Lead_Boiler] := L_Target_Setpoint;
END_IF;

// Резервный котёл: >80% или отказ основного
L_Start_Reserve :=
    L_Reserve_Available AND
    (
        (VI_Demand_Power > 80.0) OR
        (NOT L_Lead_Available)
    );

IF L_Start_Reserve THEN
    VO_Boiler_Enable[L_Reserve_Boiler] := TRUE;
    VO_Boiler_Setpoint[L_Reserve_Boiler] := L_Target_Setpoint;
END_IF;

VO_Lead_Boiler := L_Lead_Boiler;
          
END_FUNCTION_BLOCK

FUNCTION_BLOCK FB_Analog_Validator
  VAR_INPUT
    VI_Value : REAL;
    VI_Min_Valid : REAL;
    VI_Max_Valid : REAL;
    VI_Fallback_Mode : INT := 0;
    VI_Default_Value : REAL := 0.0;
  END_VAR
  VAR_OUTPUT
    VO_Value : REAL;
    VO_Error : BOOL;
  END_VAR
  VAR
    L_Last_Good_Value : REAL;
    L_First_Valid : BOOL := FALSE;
  END_VAR

            IF VI_Value >= VI_Min_Valid AND VI_Value <= VI_Max_Valid THEN
    VO_Error := FALSE;
    VO_Value := VI_Value;
    L_Last_Good_Value := VI_Value;
    L_First_Valid := TRUE;
ELSE
    VO_Error := TRUE;
    IF VI_Fallback_Mode = 1 OR NOT L_First_Valid THEN
        VO_Value := VI_Default_Value;
    ELSE
        VO_Value := L_Last_Good_Value;
    END_IF;
END_IF;
// >>> BULK_SYNC_ANCHOR: FB_Analog_Validator <<<
          
END_FUNCTION_BLOCK

FUNCTION_BLOCK FB_Sensor_Calibration_Processor
  VAR_INPUT
    VI_Raw_Value : REAL;
    VI_Record : ST_Sensor_Calibration_Record;
  END_VAR
  VAR_OUTPUT
    VO_Calibrated_Value : REAL;
  END_VAR

            VO_Calibrated_Value := (VI_Raw_Value * VI_Record.multiplier) + VI_Record.offset;
          
END_FUNCTION_BLOCK

FUNCTION_BLOCK FB_BlackBox_Recorder
  VAR_INPUT
    VI_Current_Data : ST_BlackBox_Record;
    VI_Freeze : BOOL;
  END_VAR
  VAR_OUTPUT
    VO_Frozen : BOOL;
    VO_Records_Count : INT;
  END_VAR
  VAR
    L_Write_Index : INT := 0;
    L_Initialized : BOOL := FALSE;
  END_VAR

            IF NOT L_Initialized THEN
    L_Write_Index := GVL_Retain.G_BlackBox_LastIndex;
    IF L_Write_Index < 0 OR L_Write_Index >= GVL_CONSTANTS.C_MAX_BLACKBOX_RECORDS THEN
        L_Write_Index := 0;
        GVL_Retain.G_BlackBox_LastIndex := 0;
    END_IF;
    L_Initialized := TRUE;
END_IF;

IF VI_Freeze THEN
    GVL_Retain.G_BlackBox_Frozen := TRUE;
END_IF;

VO_Frozen := GVL_Retain.G_BlackBox_Frozen;

IF NOT GVL_Retain.G_BlackBox_Frozen THEN
    GVL_Retain.G_BlackBox_Buffer[L_Write_Index] := VI_Current_Data;
    GVL_Retain.G_BlackBox_LastIndex := L_Write_Index;
    
    L_Write_Index := L_Write_Index + 1;
    IF L_Write_Index >= GVL_CONSTANTS.C_MAX_BLACKBOX_RECORDS THEN
        L_Write_Index := 0;
    END_IF;
END_IF;

VO_Records_Count := GVL_CONSTANTS.C_MAX_BLACKBOX_RECORDS; // Размер кольцевого буфера
// >>> BULK_SYNC_ANCHOR: FB_BlackBox_Recorder <<<
          
END_FUNCTION_BLOCK

FUNCTION_BLOCK FB_HMI_Interface
  VAR_INPUT
    VI_Severity : E_System_Severity;
    VI_RootCause : E_System_Root_Cause;
    VI_Status_Msg : STRING(200);
  END_VAR
  VAR_OUTPUT
    VO_HMI_Status_Text : STRING(200);
    VO_HMI_State_Code : INT;
  END_VAR

            VO_HMI_Status_Text := VI_Status_Msg;

CASE VI_Severity OF
    E_System_Severity.SEV_NORMAL:
        VO_HMI_State_Code := 0;
    E_System_Severity.SEV_WARNING:
        VO_HMI_State_Code := 1;
    E_System_Severity.SEV_DEGRADED:
        VO_HMI_State_Code := 2;
    E_System_Severity.SEV_CRITICAL:
        VO_HMI_State_Code := 3;
END_CASE;
// >>> BULK_SYNC_ANCHOR: FB_HMI_Interface <<<
          
END_FUNCTION_BLOCK

FUNCTION_BLOCK FB_Smoke_Detector
  VAR_INPUT
    VI_Smoke_Signal : BOOL;
  END_VAR
  VAR_OUTPUT
    VO_Smoke_Detected : BOOL;
  END_VAR

            VO_Smoke_Detected := VI_Smoke_Signal;
          
END_FUNCTION_BLOCK

FUNCTION_BLOCK FB_CoreKernel_Live_Observer

            
          
END_FUNCTION_BLOCK

FUNCTION_BLOCK FB_Socket_Manager
  VAR_INPUT
    VI_System_Time_MS : UDINT;
    VI_IsActivePLC : BOOL;
    VI_Scenario : E_SCENARIO_TYPE;
    VI_Fire_Alarm : BOOL;
    VI_Flood_Alarm : BOOL;
    VI_Security_Armed : BOOL;
  END_VAR
  VAR_OUTPUT
    VO_Socket_States : ARRAY[1..GVL_CONSTANTS.C_MAX_SOCKETS] OF BOOL;
    VO_Internal_States : ARRAY[1..GVL_CONSTANTS.C_MAX_SOCKETS] OF BOOL;
  END_VAR
  VAR_IN_OUT
    VI_Manual_Override : ARRAY[1..GVL_CONSTANTS.C_MAX_SOCKETS] OF BOOL;
    VI_Physical_Switches : ARRAY[1..GVL_CONSTANTS.C_MAX_SOCKETS] OF BOOL;
    VI_Rule_Actions : ARRAY[1..GVL_CONSTANTS.C_MAX_RULES] OF ST_Rule_Action;
    VI_IO_Modules_Online : ARRAY[1..GVL_CONSTANTS.C_MAX_MODULES] OF BOOL;
  END_VAR
  VAR
    fbSocketV2Staging : FB_Socket_V2_Staging;
    L_Socket_V2_Command_Shadow : ST_Socket_Command_V2;
    L_Socket_V2_State_Shadow : ST_Socket_State_V2;
    L_Socket_V2_Shadow_Diff_Found : BOOL;
    L_Socket_V2_Switch_Enabled : BOOL;
    L_Socket_V2_Path_Ready : BOOL;
    L_Socket_Using_Legacy_Fallback : BOOL;
    L_i : INT;
    L_j : INT;
    L_Rule_State : BOOL;
    L_Rule_Active : BOOL;
    L_Internal_State : ARRAY[1..GVL_CONSTANTS.C_MAX_SOCKETS] OF BOOL;
    L_Manual_Trig : ARRAY[1..GVL_CONSTANTS.C_MAX_SOCKETS] OF R_TRIG;
  END_VAR

            // Менеджер управления розетками.
// Обеспечивает работу по сценариям, правилам и аварийное отключение (без локальных выключателей розеток).


IF NOT VI_IsActivePLC THEN RETURN; END_IF;

L_Socket_V2_Shadow_Diff_Found := FALSE;
L_Socket_V2_Switch_Enabled := TRUE;
L_Socket_V2_Path_Ready := FALSE;
L_Socket_Using_Legacy_Fallback := TRUE;

// Проверка связи с модулями ввода-вывода
FOR L_i := 1 TO GVL_CONSTANTS.C_MAX_MODULES DO
    IF NOT VI_IO_Modules_Online[L_i] THEN
        // Переход в безопасное состояние при потере связи (отключение всех розеток)
        FOR L_j := 1 TO GVL_CONSTANTS.C_MAX_SOCKETS DO
            VO_Socket_States[L_j] := FALSE;
        END_FOR;
        RETURN;
    END_IF;
END_FOR;

FOR L_i := 1 TO GVL_CONSTANTS.C_MAX_SOCKETS DO
    L_Rule_Active := FALSE;
    L_Rule_State := FALSE;
    
    L_Manual_Trig[L_i](CLK := VI_Manual_Override[L_i]);
    
    // Ручное переключение
    IF L_Manual_Trig[L_i].Q THEN
        L_Internal_State[L_i] := NOT L_Internal_State[L_i];
    END_IF;

    // Проверка правил для текущей розетки
    FOR L_j := 1 TO GVL_CONSTANTS.C_MAX_RULES DO
        IF VI_Rule_Actions[L_j].Active AND VI_Rule_Actions[L_j].Target_ID = L_i THEN
            IF VI_Rule_Actions[L_j].Action_Type = E_Rule_Action_Type.ACTION_SET_SOCKET THEN
                L_Rule_Active := TRUE;
                L_Rule_State := (VI_Rule_Actions[L_j].Value > 0.5);
                L_Internal_State[L_i] := L_Rule_State; // Синхронизация внутреннего состояния
            ELSIF VI_Rule_Actions[L_j].Action_Type = E_Rule_Action_Type.ACTION_TOGGLE_SOCKET AND VI_Rule_Actions[L_j].Triggered THEN
                L_Internal_State[L_i] := NOT L_Internal_State[L_i]; // Toggle
            END_IF;
        END_IF;
    END_FOR;

    // Аварийное отключение
    IF VI_Fire_Alarm OR VI_Flood_Alarm THEN
        // Розетки 1-4 неотключаемые (холодильник, сервер и т.д.)
        IF L_i > 4 THEN
            VO_Socket_States[L_i] := FALSE;
        ELSE
            // Критические розетки сохраняют свое текущее внутреннее состояние, а не форсируются в TRUE
            VO_Socket_States[L_i] := L_Internal_State[L_i];
        END_IF;
    ELSIF VI_Scenario = E_SCENARIO_TYPE.SCENARIO_AWAY OR VI_Security_Armed THEN
        // Master Off
        IF L_i > 4 THEN
            VO_Socket_States[L_i] := FALSE;
        ELSE
            // Неотключаемые розетки могут управляться вручную
            VO_Socket_States[L_i] := L_Internal_State[L_i];
        END_IF;
    ELSE
        // Нормальный режим: состояние определяется внутренним состоянием (ручным или правилом)
        IF L_Rule_Active THEN
            VO_Socket_States[L_i] := L_Rule_State;
        ELSE
            VO_Socket_States[L_i] := L_Internal_State[L_i];
        END_IF;
    END_IF;
END_FOR;

VO_Internal_States := L_Internal_State;

// ========================================
// Socket V2 shadow execution (phase2)
// ========================================
fbSocketV2Staging(
    VI_Socket_ID := 1,
    VI_Enable := TRUE,
    VI_Target_State := VO_Socket_States[1],
    VI_Manual_Override := VI_Manual_Override[1],
    VI_Safety_Lock := (VI_Fire_Alarm OR VI_Flood_Alarm),
    VI_Scenario_ID := TO_INT(VI_Scenario),

    VI_Is_On := VO_Socket_States[1],
    VI_Manual_Override_Active := VI_Manual_Override[1],
    VI_Safety_Blocked := (VI_Fire_Alarm OR VI_Flood_Alarm),
    VI_Alarm_Active := (VI_Fire_Alarm OR VI_Flood_Alarm),

    VO_Command_Shadow => L_Socket_V2_Command_Shadow,
    VO_State_Shadow => L_Socket_V2_State_Shadow
);

// ========================================
// Socket V2 shadow validation
// ========================================
IF VO_Socket_States[1] <> L_Socket_V2_Command_Shadow.Target_State THEN
    L_Socket_V2_Shadow_Diff_Found := TRUE;
END_IF;
IF VO_Socket_States[1] <> L_Socket_V2_State_Shadow.Is_On THEN
    L_Socket_V2_Shadow_Diff_Found := TRUE;
END_IF;
IF (VI_Fire_Alarm OR VI_Flood_Alarm) <> L_Socket_V2_State_Shadow.Safety_Blocked THEN
    L_Socket_V2_Shadow_Diff_Found := TRUE;
END_IF;

// Guarded Socket V2 enable
IF L_Socket_V2_Switch_Enabled THEN
    IF NOT L_Socket_V2_Shadow_Diff_Found THEN
        L_Socket_V2_Path_Ready := TRUE;
        L_Socket_Using_Legacy_Fallback := FALSE;
    ELSE
        L_Socket_V2_Path_Ready := FALSE;
        L_Socket_Using_Legacy_Fallback := TRUE;
    END_IF;
ELSE
    L_Socket_V2_Path_Ready := FALSE;
    L_Socket_Using_Legacy_Fallback := TRUE;
END_IF;

// >>> BULK_SYNC_ANCHOR: FB_Socket_Manager <<<
          
END_FUNCTION_BLOCK

FUNCTION_BLOCK FB_Scenario_Transition_Controller
  VAR_INPUT
    VI_System_Time : UDINT;
    VI_Start_Time : UDINT;
    VI_Duration : UDINT;
    VI_Start_Value : REAL;
    VI_End_Value : REAL;
  END_VAR
  VAR_OUTPUT
    VO_Current_Value : REAL;
    VO_Transition_Done : BOOL;
  END_VAR
  VAR
    L_Elapsed : UDINT;
    L_Progress : REAL;
  END_VAR

            L_Elapsed := (SEL(VI_System_Time >= VI_Start_Time, VI_System_Time - VI_Start_Time, (4294967295 - VI_Start_Time) + VI_System_Time + 1));

IF L_Elapsed >= VI_Duration OR VI_Duration = 0 THEN
    VO_Current_Value := VI_End_Value;
    VO_Transition_Done := TRUE;
ELSE
    L_Progress := UDINT_TO_REAL(L_Elapsed) / UDINT_TO_REAL(VI_Duration);
    VO_Current_Value := VI_Start_Value + (VI_End_Value - VI_Start_Value) * L_Progress;
    VO_Transition_Done := FALSE;
END_IF;
          
END_FUNCTION_BLOCK

FUNCTION_BLOCK FB_Random_Generator
  VAR_INPUT
    VI_Seed_Value : UDINT;
  END_VAR
  VAR_INPUT
    VI_min : UDINT;
    VI_max : UDINT;
    VI_System_Time_MS : UDINT;
  END_VAR
  VAR
    L_seed : UDINT := 1;
    L_Is_Seeded : BOOL := FALSE;
  END_VAR
  VAR CONSTANT
    C_LCG_MULTIPLIER : UDINT := 1664525;
    C_LCG_INCREMENT : UDINT := 1013904223;
    C_LCG_MODULUS : LREAL := 4294967296.0;
  END_VAR
  VAR
    L_range : UDINT;
    L_rand_factor : LREAL;
  END_VAR

            
          

METHOD Seed : BOOL
                  L_seed := VI_Seed_Value;
L_Is_Seeded := TRUE;
Seed := TRUE;
                
END_METHOD

METHOD Random_Int_Range : UDINT
                  IF NOT L_Is_Seeded AND VI_System_Time_MS > 0 THEN
    L_seed := VI_System_Time_MS;
    L_Is_Seeded := TRUE;
END_IF;

L_seed := (C_LCG_MULTIPLIER * L_seed) + C_LCG_INCREMENT;

IF VI_max > VI_min THEN
        L_range := VI_max - VI_min;
        // Используем LREAL для точности и исключения выхода за границу
        L_rand_factor := TO_LREAL(L_seed) / C_LCG_MODULUS;
        Random_Int_Range := VI_min + TO_UDINT(L_rand_factor * TO_LREAL(L_range + 1));
        
        // Финальная защита от переполнения
        IF Random_Int_Range > VI_max THEN
            Random_Int_Range := VI_max;
        END_IF;
    ELSE
        Random_Int_Range := VI_min;
    END_IF;
                
END_METHOD
END_FUNCTION_BLOCK

FUNCTION_BLOCK FB_FloorHeating_Freeze_Protection
  VAR_INPUT
    VI_Outdoor_Temp : REAL;
    VI_Threshold : REAL := 7.0;
  END_VAR
  VAR_OUTPUT
    VO_Freeze_Alert : BOOL;
    VO_Pump_Force_On : BOOL;
  END_VAR
  VAR_IN_OUT
    VI_Floor_Temps : ARRAY[1..GVL_CONSTANTS.C_MAX_HEATING_CIRCUITS] OF REAL;
  END_VAR
  VAR
    L_i : INT;
  END_VAR

            VO_Freeze_Alert := FALSE;
VO_Pump_Force_On := FALSE;

FOR L_i := 1 TO GVL_CONSTANTS.C_MAX_HEATING_CIRCUITS DO
    IF VI_Floor_Temps[L_i] < VI_Threshold THEN
        VO_Freeze_Alert := TRUE;
        VO_Pump_Force_On := TRUE;
        RETURN;
    END_IF;
END_FOR;

IF VI_Outdoor_Temp < -5.0 THEN
    VO_Pump_Force_On := TRUE;
END_IF;
          
END_FUNCTION_BLOCK

FUNCTION_BLOCK FB_Trend_Logger
  VAR_INPUT
    VI_System_Time_MS : UDINT;
    VI_Config : ST_Trend_Config;
    VI_Current_Value : REAL;
  END_VAR
  VAR_OUTPUT
    VO_Data : ST_Trend_Data;
  END_VAR
  VAR
    L_Last_Log_Time : UDINT;
    L_Last_Value : REAL;
    L_Deviation : REAL;
  END_VAR

            IF NOT VI_Config.enabled THEN RETURN; END_IF;

// Логирование по изменению (Deadband) или по времени (раз в час)
L_Deviation := ABS(VI_Current_Value - L_Last_Value);
IF (L_Deviation >= (L_Last_Value * VI_Config.deviation_threshold_percent / 100.0)) OR 
   ((SEL(VI_System_Time_MS >= L_Last_Log_Time, VI_System_Time_MS - L_Last_Log_Time, (4294967295 - L_Last_Log_Time) + VI_System_Time_MS + 1)) >= GVL_CONSTANTS.C_MS_IN_HOUR) THEN
    
    // Запись в массив
    VO_Data.write_index := (VO_Data.record_count MOD 100) + 1;
    VO_Data.values[VO_Data.write_index] := VI_Current_Value;
    VO_Data.timestamps[VO_Data.write_index] := VI_System_Time_MS;

    VO_Data.record_count := VO_Data.record_count + 1;
    VO_Data.sum_values := VO_Data.sum_values + VI_Current_Value;
    
    L_Last_Value := VI_Current_Value;
    L_Last_Log_Time := VI_System_Time_MS;
END_IF;
          
END_FUNCTION_BLOCK

FUNCTION_BLOCK FB_Astro_Timer
  VAR_INPUT
    VI_System_Time_MS : UDINT;
    VI_Latitude : REAL := 55.75;
    VI_Longitude : REAL := 37.61;
    VI_Timezone : REAL := 3.0;
    VI_Day_Of_Year : UINT;
  END_VAR
  VAR_OUTPUT
    VO_Sunset_Time : TOD;
    VO_Sunrise_Time : TOD;
    VO_Is_Night : BOOL;
    VO_Current_TOD : TOD;
  END_VAR
  VAR
    L_Current_TOD : TOD;
    L_Pi : REAL := 3.14159265359;
    L_Rad : REAL := 3.14159265359 / 180.0;
    L_Deg : REAL := 180.0 / 3.14159265359;
    L_B : REAL;
    L_EoT : REAL;
    L_Declination : REAL;
    L_Cos_Omega : REAL;
    L_Omega : REAL;
    L_Sunrise_Local : REAL;
    L_Sunset_Local : REAL;
  END_VAR

            // >>> SYNC_TEST_MARKER_002 <<<


L_Current_TOD := GVL_STATUS.G_Current_TOD;
VO_Current_TOD := L_Current_TOD;

// Equation of Time (EoT) in minutes
L_B := 360.0 / 365.0 * TO_REAL(VI_Day_Of_Year - 81) * L_Rad;
L_EoT := 9.87 * SIN(2.0 * L_B) - 7.53 * COS(L_B) - 1.5 * SIN(L_B);

// Solar Declination in degrees
L_Declination := 23.45 * SIN(360.0 / 365.0 * TO_REAL(VI_Day_Of_Year + 284) * L_Rad);

// Hour angle
L_Cos_Omega := -TAN(VI_Latitude * L_Rad) * TAN(L_Declination * L_Rad);

IF L_Cos_Omega > 1.0 THEN
    L_Cos_Omega := 1.0; // Polar night
ELSIF L_Cos_Omega < -1.0 THEN
    L_Cos_Omega := -1.0; // Polar day
END_IF;

L_Omega := ACOS(L_Cos_Omega) * L_Deg;

// Sunrise and Sunset in local time (hours)
L_Sunrise_Local := 12.0 - (L_Omega / 15.0) - (L_EoT / 60.0) + (VI_Timezone * 15.0 - VI_Longitude) / 15.0;
L_Sunset_Local := 12.0 + (L_Omega / 15.0) - (L_EoT / 60.0) + (VI_Timezone * 15.0 - VI_Longitude) / 15.0;

// Handle bounds
IF L_Sunrise_Local < 0.0 THEN L_Sunrise_Local := L_Sunrise_Local + 24.0; END_IF;
IF L_Sunrise_Local >= 24.0 THEN L_Sunrise_Local := L_Sunrise_Local - 24.0; END_IF;
IF L_Sunset_Local < 0.0 THEN L_Sunset_Local := L_Sunset_Local + 24.0; END_IF;
IF L_Sunset_Local >= 24.0 THEN L_Sunset_Local := L_Sunset_Local - 24.0; END_IF;

// Конвертация в TOD
VO_Sunrise_Time := TO_TOD(TO_UDINT(L_Sunrise_Local * 3600000.0));
VO_Sunset_Time := TO_TOD(TO_UDINT(L_Sunset_Local * 3600000.0));

// ТЗ 15.2: Закат + 30 мин / Рассвет - 30 мин
VO_Is_Night := (L_Current_TOD > (VO_Sunset_Time + T#30m)) OR (L_Current_TOD < (VO_Sunrise_Time - T#30m));
// >>> SYNC_TEST_MARKER_FORCE <<<
// >>> BULK_SYNC_ANCHOR: FB_Astro_Timer <<<
          
END_FUNCTION_BLOCK

FUNCTION_BLOCK FB_Rule_Engine
  VAR_INPUT
    VI_System_Time_MS : UDINT;
    VI_IsActivePLC : BOOL;
    VI_Security_Armed : BOOL;
    VI_Current_Time : TOD;
    VI_Day_Of_Week : INT;
  END_VAR
  VAR_OUTPUT
    VO_Actions : ARRAY[1..GVL_CONSTANTS.C_MAX_RULES] OF ST_Rule_Action;
  END_VAR
  VAR_IN_OUT
    VI_Rules : ARRAY[1..GVL_CONSTANTS.C_MAX_RULES] OF ST_User_Rule;
    VI_Indoor_Temps : ARRAY[1..16] OF REAL;
    VI_Floor_Temps : ARRAY[1..8] OF REAL;
    VI_Humidities : ARRAY[1..16] OF REAL;
    VI_CO2_Levels : ARRAY[1..16] OF REAL;
    VI_Motion_Sensors : ARRAY[1..16] OF BOOL;
    VI_Door_Sensors : ARRAY[1..GVL_CONSTANTS.C_MAX_DOOR_SENSORS] OF BOOL;
    VI_Window_Sensors : ARRAY[1..16] OF BOOL;
    VI_Water_Sensors : ARRAY[1..GVL_CONSTANTS.C_MAX_FLOOD_SENSORS] OF BOOL;
    VI_Smoke_Sensors : ARRAY[1..GVL_CONSTANTS.C_MAX_SMOKE_SENSORS] OF BOOL;
    VI_Methane_Sensors : ARRAY[1..GVL_CONSTANTS.C_MAX_METHANE_SENSORS] OF REAL;
    VI_CO_Sensors : ARRAY[1..GVL_CONSTANTS.C_MAX_CO_SENSORS] OF REAL;
  END_VAR
  VAR
    L_i : INT;
    fbCompat : ARRAY[1..GVL_CONSTANTS.C_MAX_RULES] OF FB_Rule_Compatibility_Package;
    L_Compat_All_OK : BOOL;
    L_Compat_First_Warning : STRING(255);
    L_Compat_First_Warning_Latched : BOOL;
    L_Shadow_V2_Enabled : BOOL;
    L_Shadow_V2_Roundtrip_Mismatch : BOOL;
    L_Shadow_V2_First_Mismatch_Rule : INT;
    L_V2_Switch_Enabled : BOOL;
    L_V2_Path_Ready : BOOL;
    L_V2_Using_Legacy_Fallback : BOOL;
    L_Condition_Met : BOOL;
    L_Current_Value : REAL;
    L_Triggers : ARRAY[1..GVL_CONSTANTS.C_MAX_RULES] OF R_TRIG;
    L_Trigger_Count : ARRAY[1..GVL_CONSTANTS.C_MAX_RULES] OF UINT;
    L_Last_Reset_Time : UDINT;
    L_Elapsed_Time : UDINT;
  END_VAR

            IF NOT VI_IsActivePLC THEN RETURN; END_IF;

L_Compat_All_OK := TRUE;
L_Compat_First_Warning := '';
L_Compat_First_Warning_Latched := FALSE;
L_Shadow_V2_Enabled := TRUE;
L_Shadow_V2_Roundtrip_Mismatch := FALSE;
L_Shadow_V2_First_Mismatch_Rule := 0;
L_V2_Switch_Enabled := FALSE;
L_V2_Path_Ready := FALSE;
L_V2_Using_Legacy_Fallback := TRUE;

// Сброс счетчиков срабатываний каждую минуту (защита от циклических зависимостей/дребезга)
L_Elapsed_Time := (SEL(VI_System_Time_MS >= L_Last_Reset_Time, VI_System_Time_MS - L_Last_Reset_Time, (4294967295 - L_Last_Reset_Time) + VI_System_Time_MS + 1));

IF L_Elapsed_Time >= GVL_CONSTANTS.C_MS_IN_MINUTE THEN
    L_Last_Reset_Time := VI_System_Time_MS;
    FOR L_i := 1 TO GVL_CONSTANTS.C_MAX_RULES DO
        L_Trigger_Count[L_i] := 0;
    END_FOR;
END_IF;

FOR L_i := 1 TO GVL_CONSTANTS.C_MAX_RULES DO
    fbCompat[L_i](VI_Rule_Legacy := VI_Rules[L_i]);

    IF NOT fbCompat[L_i].VO_Forward_OK OR NOT fbCompat[L_i].VO_Reverse_OK THEN
        L_Compat_All_OK := FALSE;
    END_IF;

    IF (NOT L_Compat_First_Warning_Latched) AND (fbCompat[L_i].VO_Warning_Text <> '') THEN
        L_Compat_First_Warning := fbCompat[L_i].VO_Warning_Text;
        L_Compat_First_Warning_Latched := TRUE;
    END_IF;

    IF L_Shadow_V2_Enabled THEN
        IF (fbCompat[L_i].VO_Rule_Legacy_Roundtrip.Action_Type <> VI_Rules[L_i].Action_Type)
           OR (fbCompat[L_i].VO_Rule_Legacy_Roundtrip.Action_Target_ID <> VI_Rules[L_i].Action_Target_ID)
           OR (ABS(fbCompat[L_i].VO_Rule_Legacy_Roundtrip.Action_Value - VI_Rules[L_i].Action_Value) > 0.0001)
           OR (fbCompat[L_i].VO_Rule_Legacy_Roundtrip.Condition_Type <> VI_Rules[L_i].Condition_Type)
           OR (fbCompat[L_i].VO_Rule_Legacy_Roundtrip.Condition_Target_ID <> VI_Rules[L_i].Condition_Target_ID)
           OR (fbCompat[L_i].VO_Rule_Legacy_Roundtrip.Condition_Op <> VI_Rules[L_i].Condition_Op)
           OR (ABS(fbCompat[L_i].VO_Rule_Legacy_Roundtrip.Condition_Value - VI_Rules[L_i].Condition_Value) > 0.0001)
           OR (ABS(fbCompat[L_i].VO_Rule_Legacy_Roundtrip.Condition_Value_Max - VI_Rules[L_i].Condition_Value_Max) > 0.0001) THEN
            L_Shadow_V2_Roundtrip_Mismatch := TRUE;
            IF L_Shadow_V2_First_Mismatch_Rule = 0 THEN
                L_Shadow_V2_First_Mismatch_Rule := L_i;
            END_IF;
        END_IF;
    END_IF;

    // Phase 4 scaffold: optional V2 switch point.
    // Current state: always remain on legacy behavior.
    // Future state: when V2 path is implemented and validated,
    // this block becomes the controlled branch point.
    IF L_V2_Switch_Enabled AND L_V2_Path_Ready THEN
        L_V2_Using_Legacy_Fallback := FALSE;
        // V2 action-generation path placeholder.
        // No runtime behavior change yet.
    ELSE
        L_V2_Using_Legacy_Fallback := TRUE;
    END_IF;

    VO_Actions[L_i].Active := FALSE;
    IF VI_Rules[L_i].Enabled THEN
        L_Condition_Met := FALSE;
        L_Current_Value := 0.0;
        
        // Определение значения для проверки
        IF VI_Rules[L_i].Condition_Target_ID > 0 THEN
            CASE VI_Rules[L_i].Condition_Type OF
                E_Rule_Condition_Type.COND_AIR_TEMP: IF VI_Rules[L_i].Condition_Target_ID <= 16 THEN L_Current_Value := VI_Indoor_Temps[VI_Rules[L_i].Condition_Target_ID]; END_IF;
                E_Rule_Condition_Type.COND_FLOOR_TEMP: IF VI_Rules[L_i].Condition_Target_ID <= 8 THEN L_Current_Value := VI_Floor_Temps[VI_Rules[L_i].Condition_Target_ID]; END_IF;
                E_Rule_Condition_Type.COND_HUMIDITY: IF VI_Rules[L_i].Condition_Target_ID <= 16 THEN L_Current_Value := VI_Humidities[VI_Rules[L_i].Condition_Target_ID]; END_IF;
                E_Rule_Condition_Type.COND_CO2: IF VI_Rules[L_i].Condition_Target_ID <= 16 THEN L_Current_Value := VI_CO2_Levels[VI_Rules[L_i].Condition_Target_ID]; END_IF;
                E_Rule_Condition_Type.COND_MOTION: IF VI_Rules[L_i].Condition_Target_ID <= 16 THEN L_Current_Value := SEL(VI_Motion_Sensors[VI_Rules[L_i].Condition_Target_ID], 0.0, 1.0); END_IF;
                E_Rule_Condition_Type.COND_DOOR_WINDOW: 
                    IF VI_Rules[L_i].Condition_Target_ID <= GVL_CONSTANTS.C_MAX_DOOR_SENSORS THEN
                        L_Current_Value := SEL(VI_Door_Sensors[VI_Rules[L_i].Condition_Target_ID] OR VI_Window_Sensors[VI_Rules[L_i].Condition_Target_ID], 0.0, 1.0);
                    ELSIF VI_Rules[L_i].Condition_Target_ID <= 16 THEN
                        L_Current_Value := SEL(VI_Window_Sensors[VI_Rules[L_i].Condition_Target_ID], 0.0, 1.0);
                    END_IF;
                E_Rule_Condition_Type.COND_FLOOD: IF VI_Rules[L_i].Condition_Target_ID <= GVL_CONSTANTS.C_MAX_FLOOD_SENSORS THEN L_Current_Value := SEL(VI_Water_Sensors[VI_Rules[L_i].Condition_Target_ID], 0.0, 1.0); END_IF;
                E_Rule_Condition_Type.COND_SMOKE: IF VI_Rules[L_i].Condition_Target_ID <= GVL_CONSTANTS.C_MAX_SMOKE_SENSORS THEN L_Current_Value := SEL(VI_Smoke_Sensors[VI_Rules[L_i].Condition_Target_ID], 0.0, 1.0); END_IF;
                E_Rule_Condition_Type.COND_METHANE: IF VI_Rules[L_i].Condition_Target_ID <= GVL_CONSTANTS.C_MAX_METHANE_SENSORS THEN L_Current_Value := VI_Methane_Sensors[VI_Rules[L_i].Condition_Target_ID]; END_IF;
                E_Rule_Condition_Type.COND_CO: IF VI_Rules[L_i].Condition_Target_ID <= GVL_CONSTANTS.C_MAX_CO_SENSORS THEN L_Current_Value := VI_CO_Sensors[VI_Rules[L_i].Condition_Target_ID]; END_IF;
                E_Rule_Condition_Type.COND_TIME_OF_DAY: L_Current_Value := TO_REAL(TOD_TO_UDINT(VI_Current_Time) / GVL_CONSTANTS.C_MS_IN_MINUTE); // Время в минутах
                E_Rule_Condition_Type.COND_DAY_OF_WEEK: L_Current_Value := TO_REAL(VI_Day_Of_Week);
            END_CASE;
        ELSE
            IF VI_Rules[L_i].Condition_Type = E_Rule_Condition_Type.COND_TIME_OF_DAY THEN
                L_Current_Value := TO_REAL(TOD_TO_UDINT(VI_Current_Time) / GVL_CONSTANTS.C_MS_IN_MINUTE); // Время в минутах
            ELSIF VI_Rules[L_i].Condition_Type = E_Rule_Condition_Type.COND_DAY_OF_WEEK THEN
                L_Current_Value := TO_REAL(VI_Day_Of_Week);
            END_IF;
        END_IF;
        
        // Проверка условия
        CASE VI_Rules[L_i].Condition_Op OF
            E_Rule_Comparison.COMP_GT: L_Condition_Met := (L_Current_Value > VI_Rules[L_i].Condition_Value);
            E_Rule_Comparison.COMP_LT: L_Condition_Met := (L_Current_Value < VI_Rules[L_i].Condition_Value);
            E_Rule_Comparison.COMP_EQ: L_Condition_Met := (ABS(L_Current_Value - VI_Rules[L_i].Condition_Value) < 0.1);
            E_Rule_Comparison.COMP_GE: L_Condition_Met := (L_Current_Value >= VI_Rules[L_i].Condition_Value);
            E_Rule_Comparison.COMP_LE: L_Condition_Met := (L_Current_Value <= VI_Rules[L_i].Condition_Value);
            E_Rule_Comparison.COMP_IN_RANGE: L_Condition_Met := (L_Current_Value >= VI_Rules[L_i].Condition_Value) AND (L_Current_Value <= VI_Rules[L_i].Condition_Value_Max);
            E_Rule_Comparison.COMP_TRUE: L_Condition_Met := (L_Current_Value > 0.5);
            E_Rule_Comparison.COMP_FALSE: L_Condition_Met := (L_Current_Value < 0.5);
        END_CASE;
        
        // Формирование действия
        L_Triggers[L_i](CLK := L_Condition_Met);
        
        IF L_Triggers[L_i].Q THEN
            L_Trigger_Count[L_i] := L_Trigger_Count[L_i] + 1;
            IF L_Trigger_Count[L_i] > 10 THEN
                // ТЗ 13.5: Блокировка правила при слишком частом срабатывании (циклическая зависимость)
                VO_Actions[L_i].Active := FALSE;
                VO_Actions[L_i].Triggered := FALSE;
                CONTINUE; // Пропускаем выполнение
            END_IF;
        END_IF;
        
        IF L_Condition_Met AND (L_Trigger_Count[L_i] <= 10) THEN
            VO_Actions[L_i].Active := TRUE;
            VO_Actions[L_i].Triggered := L_Triggers[L_i].Q;
            VO_Actions[L_i].Action_Type := VI_Rules[L_i].Action_Type;
            VO_Actions[L_i].Target_ID := VI_Rules[L_i].Action_Target_ID;
            VO_Actions[L_i].Value := VI_Rules[L_i].Action_Value;
        END_IF;
    END_IF;
END_FOR;
// >>> BULK_SYNC_ANCHOR: FB_Rule_Engine <<<
          
END_FUNCTION_BLOCK

FUNCTION_BLOCK FB_Command_Deduplication
  VAR_INPUT
    VI_Command_ID : UDINT;
    VI_Command_Type : E_Gateway_Command_Type;
    VI_Command_Value : REAL;
    VI_System_Time_MS : UDINT;
  END_VAR
  VAR_OUTPUT
    VO_Is_New_Command : BOOL;
    VO_Processed_ID : UDINT;
  END_VAR
  VAR
    L_Processed_History : ARRAY[0..GVL_CONSTANTS.C_MAX_DEDUPLICATION_HISTORY-1] OF UDINT;
    L_Processed_Times : ARRAY[0..GVL_CONSTANTS.C_MAX_DEDUPLICATION_HISTORY-1] OF UDINT;
    L_History_Index : INT := 0;
    L_i : INT;
    L_Found : BOOL;
  END_VAR

            // Check if command ID is already in history
L_Found := FALSE;
FOR L_i := 0 TO GVL_CONSTANTS.C_MAX_DEDUPLICATION_HISTORY-1 DO
    IF L_Processed_History[L_i] = VI_Command_ID AND VI_Command_ID <> 0 THEN
        // Check if the command is not too old (e.g., 1 hour = 3600000 ms)
        IF (VI_System_Time_MS - L_Processed_Times[L_i]) < 3600000 THEN
            L_Found := TRUE;
            EXIT;
        END_IF;
    END_IF;
END_FOR;

IF NOT L_Found AND VI_Command_ID <> 0 THEN
    // New command detected
    VO_Is_New_Command := TRUE;
    VO_Processed_ID := VI_Command_ID;
    
    // Add to history
    L_Processed_History[L_History_Index] := VI_Command_ID;
    L_Processed_Times[L_History_Index] := VI_System_Time_MS;
    L_History_Index := L_History_Index + 1;
    IF L_History_Index > GVL_CONSTANTS.C_MAX_DEDUPLICATION_HISTORY-1 THEN
        L_History_Index := 0;
    END_IF;
ELSE
    // Duplicate or empty command
    VO_Is_New_Command := FALSE;
    VO_Processed_ID := 0;
END_IF;
          
END_FUNCTION_BLOCK

FUNCTION_BLOCK FB_Water_Leakage_Manager
  VAR_INPUT
    VI_System_Time_MS : UDINT;
    VI_IsActivePLC : BOOL;
    VI_Config : ST_Flood_Global_Config;
  END_VAR
  VAR_OUTPUT
    VO_Close_Valve_35 : BOOL;
    VO_Close_Valve_36 : BOOL;
    VO_Status_Msg : STRING(200);
    VO_Leak_Detected : BOOL;
    VO_Leak_Warning_Level : BOOL;
  END_VAR
  VAR_IN_OUT
    VI_Sensors : ARRAY[1..GVL_CONSTANTS.C_MAX_FLOOD_SENSORS] OF BOOL;
  END_VAR
  VAR
    L_i : INT;
    L_Sensor_Timers : ARRAY[1..GVL_CONSTANTS.C_MAX_FLOOD_SENSORS] OF FB_System_Timer;
    L_Any_Leak : BOOL;
    L_Any_Warning : BOOL;
  END_VAR

            IF NOT VI_IsActivePLC THEN RETURN; END_IF;

L_Any_Leak := FALSE;
L_Any_Warning := FALSE;

FOR L_i := 1 TO GVL_CONSTANTS.C_MAX_FLOOD_SENSORS DO
    L_Sensor_Timers[L_i](
        IN := VI_Sensors[L_i],
        PT := TO_TIME(VI_Config.min_duration_ms + VI_Config.warning_duration_ms),
        VI_System_Time_MS := VI_System_Time_MS
    );

    IF L_Sensor_Timers[L_i].ET >= TO_TIME(VI_Config.min_duration_ms) THEN
        L_Any_Warning := TRUE;

        IF L_Sensor_Timers[L_i].Q THEN
            L_Any_Leak := TRUE;

            IF VI_Config.sensor_to_valve_map[L_i] = 1 THEN
                VO_Close_Valve_35 := TRUE;
            ELSIF VI_Config.sensor_to_valve_map[L_i] = 2 THEN
                VO_Close_Valve_36 := TRUE;
            END_IF;
        END_IF;
    END_IF;
END_FOR;

// Health signals
VO_Leak_Detected := L_Any_Leak;
VO_Leak_Warning_Level := L_Any_Warning;

// Status
IF L_Any_Leak THEN
    VO_Status_Msg := 'АВАРИЯ: ПРОТЕЧКА ВОДЫ. КЛАПАНЫ ЗАКРЫТЫ.';
ELSIF L_Any_Warning THEN
    VO_Status_Msg := 'ПРЕДУПРЕЖДЕНИЕ: ОБНАРУЖЕНА ВОДА.';
ELSE
    VO_Status_Msg := 'Система контроля протечек в норме';
    VO_Close_Valve_35 := FALSE;
    VO_Close_Valve_36 := FALSE;
END_IF;
// >>> BULK_SYNC_ANCHOR: FB_Water_Leakage_Manager <<<
          
END_FUNCTION_BLOCK

FUNCTION_BLOCK FB_State_Manager_MVP
  VAR_INPUT
    VI_Gas_Alarm : BOOL;
    VI_Fire_Alarm : BOOL;
    VI_Flood_Alarm : BOOL;
    VI_IO_Healthy : BOOL;
    VI_Freeze_Risk : BOOL;
    VI_Reset_Request : BOOL;
  END_VAR
  VAR_OUTPUT
    VO_System_Mode : INT;
  END_VAR
  VAR
    L_Fire_Latched : BOOL;
    L_Gas_Latched : BOOL;
    L_Flood_Latched : BOOL;
  END_VAR

            FUNCTION_BLOCK FB_State_Manager


// Fire latch
IF VI_Fire_Alarm THEN
    L_Fire_Latched := TRUE;
END_IF;
IF VI_Reset_Request AND NOT VI_Fire_Alarm THEN
    L_Fire_Latched := FALSE;
END_IF;

// Gas latch
IF VI_Gas_Alarm THEN
    L_Gas_Latched := TRUE;
END_IF;
IF VI_Reset_Request AND NOT VI_Gas_Alarm THEN
    L_Gas_Latched := FALSE;
END_IF;

// Flood latch
IF VI_Flood_Alarm THEN
    L_Flood_Latched := TRUE;
END_IF;
IF VI_Reset_Request AND NOT VI_Flood_Alarm THEN
    L_Flood_Latched := FALSE;
END_IF;

// Mode logic
IF L_Fire_Latched THEN
    VO_System_Mode := 2; // SAFE_STOP
ELSIF L_Flood_Latched THEN
    VO_System_Mode := 2;
ELSIF L_Gas_Latched THEN
    IF VI_Freeze_Risk THEN
        VO_System_Mode := 3; // FREEZE
    ELSE
        VO_System_Mode := 1; // DEGRADED
    END_IF;
ELSIF NOT VI_IO_Healthy THEN
    VO_System_Mode := 1;
ELSE
    VO_System_Mode := 0; // NORMAL
END_IF;
          
END_FUNCTION_BLOCK

FUNCTION_BLOCK FB_Ventilation_System_Manager
  VAR_INPUT
    VI_System_Time_MS : UDINT;
    VI_IsActivePLC : BOOL;
    VI_Outdoor_Temp : REAL;
    VI_Current_Scenario : E_SCENARIO_TYPE;
    VI_System_Mode : E_System_Operating_Mode;
    VI_Config : ST_Ventilation_Global_Config;
    VI_Fire_Alarm : BOOL;
    VI_Gas_Alarm : BOOL;
    VI_PV3_Boost_Req : BOOL;
    VI_Supply_100_Req : BOOL;
    VI_Exhaust_100_Req : BOOL;
    VI_Supply_80_Req : BOOL;
    VI_Vent_Stop : BOOL;
    VI_IO_Modules_Online : ARRAY[1..GVL_CONSTANTS.C_MAX_MODULES] OF BOOL;
  END_VAR
  VAR_OUTPUT
    VO_Supply_Fans : ARRAY[1..GVL_CONSTANTS.C_MAX_SUPPLY_FANS] OF BYTE;
    VO_Exhaust_Fans : ARRAY[1..GVL_CONSTANTS.C_MAX_EXHAUST_FANS] OF BYTE;
    VO_Heater_Power : ARRAY[1..GVL_CONSTANTS.C_MAX_BOILERS] OF REAL;
    VO_Status_Msg : STRING(200);
  END_VAR
  VAR_IN_OUT
    VI_Supply_Temps : ARRAY[1..GVL_CONSTANTS.C_MAX_SUPPLY_TEMPS] OF REAL;
    VI_Room_Temps : ARRAY[1..16] OF REAL;
    VI_Room_Humidities : ARRAY[1..16] OF REAL;
    VI_Room_CO2 : ARRAY[1..16] OF REAL;
    VI_Wet_Zone_Active : ARRAY[1..GVL_CONSTANTS.C_MAX_WET_ZONES] OF BOOL;
    VI_Rule_Actions : ARRAY[1..GVL_CONSTANTS.C_MAX_RULES] OF ST_Rule_Action;
  END_VAR
  VAR
    L_Policy_Normal : BOOL;
    L_Policy_Safe_Stop : BOOL;
    L_Policy_Degraded : BOOL;
    L_Policy_Freeze_Protection : BOOL;
    L_i : INT;
    L_j : INT;
    L_Max_CO2 : REAL;
    L_Max_Hum : REAL;
    L_Base_Speed : BYTE;
    L_Target_Temp : REAL;
    L_PID_Heaters : ARRAY[1..GVL_CONSTANTS.C_MAX_BOILERS] OF FB_PID_Controller;
    L_Wet_Zone_Timers : ARRAY[1..GVL_CONSTANTS.C_MAX_WET_ZONES] OF FB_System_Timer_TOF;
    fbVentilationV2Staging : FB_Ventilation_V2_Staging;
    L_Vent_Command_Shadow : ST_Ventilation_Command_V2;
    L_Vent_State_Shadow : ST_Ventilation_State_V2;
    L_Vent_V2_Shadow_Diff_Found : BOOL;
    L_Vent_V2_Switch_Enabled : BOOL;
    L_Vent_V2_Path_Ready : BOOL;
    L_Vent_Using_Legacy_Fallback : BOOL;
  END_VAR

            // ========================================
// Ventilation policy layer (phase3/v2)
// ========================================
GVL_STATE.G_Ventilation_IO_Fault := FALSE;
GVL_STATE.G_Ventilation_Subsystem_Degraded := FALSE;
L_Vent_V2_Shadow_Diff_Found := FALSE;
L_Vent_V2_Switch_Enabled := TRUE;
L_Vent_V2_Path_Ready := FALSE;
L_Vent_Using_Legacy_Fallback := TRUE;
L_Policy_Normal := (VI_System_Mode = E_System_Operating_Mode.MODE_NORMAL);
L_Policy_Safe_Stop := (VI_System_Mode = E_System_Operating_Mode.MODE_SAFE_STOP);
L_Policy_Degraded := (VI_System_Mode = E_System_Operating_Mode.MODE_DEGRADED);
L_Policy_Freeze_Protection := (VI_System_Mode = E_System_Operating_Mode.MODE_FREEZE_PROTECTION);

IF NOT VI_IsActivePLC THEN
    FOR L_i := 1 TO GVL_CONSTANTS.C_MAX_SUPPLY_FANS DO
        VO_Supply_Fans[L_i] := 0;
        IF L_i <= GVL_CONSTANTS.C_MAX_SUPPLY_TEMPS THEN
            VO_Heater_Power[L_i] := 0.0;
        END_IF;
    END_FOR;
    FOR L_i := 1 TO GVL_CONSTANTS.C_MAX_EXHAUST_FANS DO
        VO_Exhaust_Fans[L_i] := 0;
    END_FOR;
    VO_Status_Msg := 'ВЕНТИЛЯЦИЯ: РЕЗЕРВНЫЙ ПЛК';
    RETURN;
END_IF;

// Проверка связи с модулями ввода-вывода
FOR L_i := 1 TO GVL_CONSTANTS.C_MAX_MODULES DO
    IF NOT VI_IO_Modules_Online[L_i] THEN
        GVL_STATE.G_Ventilation_IO_Fault := TRUE;
        // Переход в безопасное состояние при потере связи (отключение вентиляции)
        FOR L_j := 1 TO GVL_CONSTANTS.C_MAX_SUPPLY_FANS DO
            VO_Supply_Fans[L_j] := 0;
        END_FOR;
        FOR L_j := 1 TO GVL_CONSTANTS.C_MAX_EXHAUST_FANS DO
            VO_Exhaust_Fans[L_j] := 0;
        END_FOR;
        FOR L_j := 1 TO GVL_CONSTANTS.C_MAX_BOILERS DO
            VO_Heater_Power[L_j] := 0.0;
        END_FOR;
        VO_Status_Msg := 'ОШИБКА: Потеря связи с модулями ввода-вывода';
        RETURN;
    END_IF;
END_FOR;

// =========================
// SYSTEM MODE OVERRIDE
// =========================
// VENT_POLICY_ROUTING_PHASE3_V2
IF L_Policy_Safe_Stop THEN
    FOR L_i := 1 TO GVL_CONSTANTS.C_MAX_SUPPLY_FANS DO
        VO_Supply_Fans[L_i] := 0;
    END_FOR;
    FOR L_i := 1 TO GVL_CONSTANTS.C_MAX_EXHAUST_FANS DO
        VO_Exhaust_Fans[L_i] := 0;
    END_FOR;
    FOR L_i := 1 TO GVL_CONSTANTS.C_MAX_BOILERS DO
        VO_Heater_Power[L_i] := 0.0;
    END_FOR;
    VO_Status_Msg := 'ВЕНТИЛЯЦИЯ: ОСТАНОВЛЕНА POLICY SAFE_STOP';
    RETURN;
END_IF;

IF L_Policy_Degraded THEN
    FOR L_i := 1 TO GVL_CONSTANTS.C_MAX_SUPPLY_FANS DO
        VO_Supply_Fans[L_i] := 0;
    END_FOR;
    FOR L_i := 1 TO GVL_CONSTANTS.C_MAX_BOILERS DO
        VO_Heater_Power[L_i] := 0.0;
    END_FOR;
    GVL_STATE.G_Ventilation_Subsystem_Degraded := TRUE;
    VO_Status_Msg := 'ВЕНТИЛЯЦИЯ: DEGRADED POLICY';
END_IF;

IF L_Policy_Freeze_Protection THEN
    FOR L_i := 1 TO GVL_CONSTANTS.C_MAX_SUPPLY_FANS DO
        VO_Supply_Fans[L_i] := 0;
    END_FOR;
    FOR L_i := 1 TO GVL_CONSTANTS.C_MAX_EXHAUST_FANS DO
        VO_Exhaust_Fans[L_i] := 0;
    END_FOR;
    FOR L_i := 1 TO GVL_CONSTANTS.C_MAX_BOILERS DO
        VO_Heater_Power[L_i] := 0.0;
    END_FOR;
    VO_Status_Msg := 'ВЕНТИЛЯЦИЯ: FREEZE_PROTECTION POLICY (stop)';
    RETURN;
END_IF;

// MODE_FREEZE_PROTECTION пока оставляем на текущей штатной логике

// 1. Определение базовой скорости и целевой температуры по сценарию (ТЗ 7.1)
CASE VI_Current_Scenario OF
    E_SCENARIO_TYPE.SCENARIO_AWAY:
        L_Base_Speed := VI_Config.Scenario_Modes[3].Base_Fan_Speed;
        L_Target_Temp := VI_Config.Scenario_Modes[3].Target_Temp;
    E_SCENARIO_TYPE.SCENARIO_SLEEP:
        L_Base_Speed := VI_Config.Scenario_Modes[2].Base_Fan_Speed;
        L_Target_Temp := VI_Config.Scenario_Modes[2].Target_Temp;
    ELSE // PRESENCE, MORNING, EVENING
        L_Base_Speed := VI_Config.Scenario_Modes[1].Base_Fan_Speed;
        L_Target_Temp := VI_Config.Scenario_Modes[1].Target_Temp;
END_CASE;

// 2. Логика управления приточными установками (П-1, П-2, П-3)
FOR L_i := 1 TO GVL_CONSTANTS.C_MAX_SUPPLY_FANS DO
    // ПИД-регулирование мощности электрического калорифера
    IF L_i <= GVL_CONSTANTS.C_MAX_SUPPLY_TEMPS THEN
        L_PID_Heaters[L_i](
            VI_SetPoint := L_Target_Temp,
            VI_ProcessValue := VI_Supply_Temps[L_i], // Используем датчик температуры после калорифера
            VI_Kp := 4.0, VI_Tn := 120.0, VI_Tv := 0.0,
            VI_Y_Min := 0.0, VI_Y_Max := 100.0, VI_Cycle_Time_S := 1.0,
            VO_Output => VO_Heater_Power[L_i]
        );
    END_IF;

    // Определение скорости приточного вентилятора
    VO_Supply_Fans[L_i] := L_Base_Speed;
    
    // Обработка действий от Rule Engine
    FOR L_j := 1 TO GVL_CONSTANTS.C_MAX_RULES DO
        IF VI_Rule_Actions[L_j].Active AND VI_Rule_Actions[L_j].Target_ID = L_i THEN
            IF VI_Rule_Actions[L_j].Action_Type = E_Rule_Action_Type.ACTION_SET_VENTILATION THEN
                VO_Supply_Fans[L_i] := REAL_TO_BYTE(VI_Rule_Actions[L_j].Value);
            END_IF;
        END_IF;
    END_FOR;
    
    // Requests are observed but must not bypass policy directly.
    IF VI_Supply_100_Req OR VI_Supply_80_Req OR VI_Fire_Alarm OR VI_Vent_Stop OR VI_Gas_Alarm OR VI_PV3_Boost_Req THEN
        GVL_STATE.G_Ventilation_Subsystem_Degraded := TRUE;
    END_IF;
END_FOR;

// 3. Логика управления вытяжными установками (В-1 .. В-5)
FOR L_i := 1 TO GVL_CONSTANTS.C_MAX_EXHAUST_FANS DO
    VO_Exhaust_Fans[L_i] := L_Base_Speed;
    
    // ТЗ 4.0: Логика вытяжки в санузлах
    FOR L_j := 1 TO GVL_CONSTANTS.C_MAX_WET_ZONES DO
        IF VI_Config.wet_zone_to_exhaust_map[L_j] = L_i THEN
            // Включение по свету, выключение с задержкой 5 минут (используем TOF)
            L_Wet_Zone_Timers[L_j](IN := VI_Wet_Zone_Active[L_j], PT := T#5m, VI_System_Time_MS := VI_System_Time_MS);
            IF VI_Wet_Zone_Active[L_j] THEN
                VO_Exhaust_Fans[L_i] := 80; // Повышенная скорость при присутствии
            ELSIF L_Wet_Zone_Timers[L_j].Q THEN
                VO_Exhaust_Fans[L_i] := 50; // Скорость выбега (пока таймер TOF активен)
            END_IF;
        END_IF;
    END_FOR;

    // Requests are observed but must not bypass policy directly.
    IF (L_i = VI_Config.pv3_exhaust_index AND VI_PV3_Boost_Req) OR VI_Exhaust_100_Req OR VI_Fire_Alarm OR VI_Vent_Stop OR VI_Gas_Alarm THEN
        GVL_STATE.G_Ventilation_Subsystem_Degraded := TRUE;
    END_IF;
END_FOR;








// ========================================
// VENT_FINAL_CLAMP
// ========================================
IF L_Policy_Degraded THEN
    FOR L_i := 1 TO GVL_CONSTANTS.C_MAX_EXHAUST_FANS DO
        VO_Exhaust_Fans[L_i] := MIN(VO_Exhaust_Fans[L_i], VI_Config.Degraded_Exhaust_Limit);
    END_FOR;
END_IF;

// Ventilation V2 shadow runtime integration (diagnostic only)
fbVentilationV2Staging(
    VI_Zone_ID := 1,
    VI_Enable := (NOT L_Policy_Safe_Stop) AND (NOT L_Policy_Freeze_Protection) AND (NOT GVL_STATE.G_Ventilation_IO_Fault),
    VI_Fan_Speed_Setpoint := BYTE_TO_REAL(VO_Supply_Fans[1]),
    VI_Damper_Position_Setpoint := 0.0,
    VI_Heat_Recovery_Enabled := L_Policy_Normal,
    VI_Is_Active := (VO_Supply_Fans[1] > 0) OR (VO_Exhaust_Fans[1] > 0),
    VI_Fan_Speed_Actual := BYTE_TO_REAL(VO_Supply_Fans[1]),
    VI_Supply_Temp := VI_Supply_Temps[1],
    VI_Extract_Temp := VI_Room_Temps[1],
    VI_Filter_Dirty := FALSE,
    VI_Alarm_Active := GVL_STATE.G_Ventilation_IO_Fault OR GVL_STATE.G_Ventilation_Subsystem_Degraded,
    VO_Command_Shadow => L_Vent_Command_Shadow,
    VO_State_Shadow => L_Vent_State_Shadow
);

// Ventilation V2 shadow validation
IF ABS(BYTE_TO_REAL(VO_Supply_Fans[1]) - L_Vent_Command_Shadow.Fan_Speed_Setpoint) > 0.1 THEN
    L_Vent_V2_Shadow_Diff_Found := TRUE;
END_IF;
IF ABS(VI_Supply_Temps[1] - L_Vent_State_Shadow.Supply_Temp) > 0.1 THEN
    L_Vent_V2_Shadow_Diff_Found := TRUE;
END_IF;

